LIN {X 0,Y 179.244,Z 433.398,A -85,B 0,C 180,E1 -24811.852,E2 -24811.852} C_VEL
LIN {X 0,Y 175.671,Z 428.049,A -85,B 0,C 180,E1 -24814.607,E2 -24814.607} C_VEL
LIN {X 0,Y 173.718,Z 425.111,A -85,B 0,C 180,E1 -24816.292,E2 -24816.292} C_VEL
LIN {X 0,Y 171.255,Z 421.543,A -85,B 0,C 180,E1 -24818.641,E2 -24818.641} C_VEL
LIN {X 0,Y 168.544,Z 417.832,A -85,B 0,C 180,E1 -24821.618,E2 -24821.618} C_VEL
LIN {X 0,Y 167.606,Z 416.657,A -85,B 0,C 180,E1 -24822.774,E2 -24822.774} C_VEL
LIN {X 0,Y 165.097,Z 413.195,A -85,B 0,C 180,E1 -24826.459,E2 -24826.459} C_VEL
LIN {X 0,Y 164.62,Z 412.184,A -85,B 0,C 180,E1 -24827.361,E2 -24827.361} C_VEL
LIN {X 0,Y 161.279,Z 407.116,A -85,B 0,C 180,E1 -24838.751,E2 -24838.751} C_VEL
LIN {X 0,Y 161.263,Z 406.995,A -85,B 0,C 180,E1 -24840.624,E2 -24840.624} C_VEL
LIN {X 0,Y 161.713,Z 408.835,A -85,B 0,C 180,E1 -24845.299,E2 -24845.299} C_VEL
LIN {X 0,Y 164.838,Z 412.58,A -85,B 0,C 180,E1 -24853.091,E2 -24853.091} C_VEL
LIN {X 0,Y 167.223,Z 416.316,A -85,B 0,C 180,E1 -24856.794,E2 -24856.794} C_VEL
LIN {X 0,Y 168.452,Z 417.684,A -85,B 0,C 180,E1 -24858.313,E2 -24858.313} C_VEL
LIN {X 0,Y 171.212,Z 421.521,A -85,B 0,C 180,E1 -24861.365,E2 -24861.365} C_VEL
LIN {X 0,Y 175.071,Z 427.086,A -85,B 0,C 180,E1 -24864.93,E2 -24864.93} C_VEL
LIN {X 0,Y 179.814,Z 434.296,A -85,B 0,C 180,E1 -24868.604,E2 -24868.604} C_VEL
LIN {X 0,Y 184.893,Z 442.842,A -85,B 0,C 180,E1 -24871.99,E2 -24871.99} C_VEL
LIN {X 0,Y 189.293,Z 452.81,A -85,B 0,C 180,E1 -24874.721,E2 -24874.721} C_VEL
LIN {X 0,Y 191.912,Z 459.666,A -85,B 0,C 180,E1 -24876.262,E2 -24876.262} C_VEL
LIN {X 0,Y 188.369,Z 504.662,A -85,B 0,C 180,E1 -24877.636,E2 -24877.636} C_VEL
LIN {X 0,Y 186.538,Z 518.919,A -85,B 0,C 180,E1 -24878.256,E2 -24878.256} C_VEL
LIN {X 0,Y 183.633,Z 533.235,A -85,B 0,C 180,E1 -24879.199,E2 -24879.199} C_VEL
LIN {X 0,Y 180.047,Z 546.434,A -85,B 0,C 180,E1 -24880.438,E2 -24880.438} C_VEL
LIN {X 0,Y 176.027,Z 558.458,A -85,B 0,C 180,E1 -24881.965,E2 -24881.965} C_VEL
LIN {X 0,Y 171.04,Z 570.911,A -85,B 0,C 180,E1 -24884.027,E2 -24884.027} C_VEL
LIN {X 0,Y 167.715,Z 578.171,A -85,B 0,C 180,E1 -24885.532,E2 -24885.532} C_VEL
LIN {X 0,Y 165.051,Z 582.747,A -85,B 0,C 180,E1 -24886.466,E2 -24886.466} C_VEL
LIN {X 0,Y 159.051,Z 589.893,A -85,B 0,C 180,E1 -24887.711,E2 -24887.711} C_VEL
LIN {X 0,Y 152.884,Z 596.609,A -85,B 0,C 180,E1 -24889.164,E2 -24889.164} C_VEL
LIN {X 0,Y 149.983,Z 600.384,A -85,B 0,C 180,E1 -24890.442,E2 -24890.442} C_VEL
LIN {X 0,Y 144.381,Z 608.729,A -85,B 0,C 180,E1 -24894.264,E2 -24894.264} C_VEL
LIN {X 0,Y 139.661,Z 615.209,A -85,B 0,C 180,E1 -24898.109,E2 -24898.109} C_VEL
LIN {X 0,Y 135.799,Z 620.586,A -85,B 0,C 180,E1 -24902.244,E2 -24902.244} C_VEL
LIN {X 0,Y 131.508,Z 626.247,A -85,B 0,C 180,E1 -24908.036,E2 -24908.036} C_VEL
LIN {X 0,Y 128.509,Z 630.353,A -85,B 0,C 180,E1 -24914.135,E2 -24914.135} C_VEL
LIN {X 0,Y 126.82,Z 633.026,A -85,B 0,C 180,E1 -24920.434,E2 -24920.434} C_VEL
LIN {X 0,Y 126.305,Z 634.341,A -85,B 0,C 180,E1 -24926.814,E2 -24926.814} C_VEL
LIN {X 0,Y 126.32,Z 634.5,A -85,B 0,C 180,E1 -24930.004,E2 -24930.004} C_VEL
LIN {X 0,Y 126.492,Z 633.821,A -85,B 0,C 180,E1 -24936.384,E2 -24936.384} C_VEL
LIN {X 0,Y 127.846,Z 631.805,A -85,B 0,C 180,E1 -24942.707,E2 -24942.707} C_VEL
LIN {X 0,Y 130.668,Z 628.407,A -85,B 0,C 180,E1 -24948.831,E2 -24948.831} C_VEL
LIN {X 0,Y 133.685,Z 625.344,A -85,B 0,C 180,E1 -24952.918,E2 -24952.918} C_VEL
LIN {X 0,Y 137.389,Z 628.317,A -85,B 0,C 180,E1 -24957.416,E2 -24957.416} C_VEL
LIN {X 0,Y 143.434,Z 631.102,A -85,B 0,C 180,E1 -24962.618,E2 -24962.618} C_VEL
LIN {X 0,Y 151.002,Z 632.815,A -85,B 0,C 180,E1 -24967.236,E2 -24967.236} C_VEL
LIN {X 0,Y 159.895,Z 633.459,A -85,B 0,C 180,E1 -24971.251,E2 -24971.251} C_VEL
LIN {X 0,Y 169.8,Z 633.01,A -85,B 0,C 180,E1 -24974.722,E2 -24974.722} C_VEL
LIN {X 0,Y 171.46,Z 632.84,A -85,B 0,C 180,E1 -24975.828,E2 -24975.828} C_VEL
LIN {X 0,Y 161.323,Z 633.521,A -85,B 0,C 180,E1 -24979.196,E2 -24979.196} C_VEL
LIN {X 0,Y 152.228,Z 633.038,A -85,B 0,C 180,E1 -24983.118,E2 -24983.118} C_VEL
LIN {X 0,Y 144.519,Z 631.444,A -85,B 0,C 180,E1 -24987.661,E2 -24987.661} C_VEL
LIN {X 0,Y 138.231,Z 628.727,A -85,B 0,C 180,E1 -24992.769,E2 -24992.769} C_VEL
LIN {X 0,Y 133.649,Z 624.844,A -85,B 0,C 180,E1 -24998.402,E2 -24998.402} C_VEL
LIN {X 0,Y 130.688,Z 619.649,A -85,B 0,C 180,E1 -25004.402,E2 -25004.402} C_VEL
LIN {X 0,Y 129.529,Z 613.033,A -85,B 0,C 180,E1 -25010.632,E2 -25010.632} C_VEL
LIN {X 0,Y 129.643,Z 606.868,A -85,B 0,C 180,E1 -25015.336,E2 -25015.336} C_VEL
LIN {X 0,Y 129.888,Z 600.509,A -85,B 0,C 180,E1 -25019.225,E2 -25019.225} C_VEL
LIN {X 0,Y 129.965,Z 592.706,A -85,B 0,C 180,E1 -25023.1,E2 -25023.1} C_VEL
LIN {X 0,Y 130.141,Z 583.047,A -85,B 0,C 180,E1 -25026.979,E2 -25026.979} C_VEL
LIN {X 0,Y 130.686,Z 571.183,A -85,B 0,C 180,E1 -25030.849,E2 -25030.849} C_VEL
LIN {X 0,Y 131.008,Z 565.155,A -85,B 0,C 180,E1 -25032.705,E2 -25032.705} C_VEL
LIN {X 0,Y 130.969,Z 564.229,A -85,B 0,C 180,E1 -25033.527,E2 -25033.527} C_VEL
LIN {X 0,Y 131.194,Z 564.312,A -85,B 0,C 180,E1 -25034.387,E2 -25034.387} C_VEL
LIN {X 0,Y 132.105,Z 563.892,A -85,B 0,C 180,E1 -25035.427,E2 -25035.427} C_VEL
LIN {X 0,Y 133.005,Z 563.215,A -85,B 0,C 180,E1 -25036.124,E2 -25036.124} C_VEL
LIN {X 0,Y 134.669,Z 561.654,A -85,B 0,C 180,E1 -25037.08,E2 -25037.08} C_VEL
LIN {X 0,Y 135.986,Z 560.715,A -85,B 0,C 180,E1 -25038.065,E2 -25038.065} C_VEL
LIN {X 0,Y 137.57,Z 559.906,A -85,B 0,C 180,E1 -25039.4,E2 -25039.4} C_VEL
LIN {X 0,Y 139.56,Z 558.421,A -85,B 0,C 180,E1 -25040.641,E2 -25040.641} C_VEL
LIN {X 0,Y 142.131,Z 555.895,A -85,B 0,C 180,E1 -25041.769,E2 -25041.769} C_VEL
LIN {X 0,Y 144.345,Z 554.176,A -85,B 0,C 180,E1 -25042.924,E2 -25042.924} C_VEL
LIN {X 0,Y 146.147,Z 552.999,A -85,B 0,C 180,E1 -25043.973,E2 -25043.973} C_VEL
LIN {X 0,Y 149.832,Z 549.473,A -85,B 0,C 180,E1 -25045.449,E2 -25045.449} C_VEL
LIN {X 0,Y 154.004,Z 544.288,A -85,B 0,C 180,E1 -25046.63,E2 -25046.63} C_VEL
LIN {X 0,Y 157.396,Z 541.143,A -85,B 0,C 180,E1 -25047.96,E2 -25047.96} C_VEL
LIN {X 0,Y 160.767,Z 537.171,A -85,B 0,C 180,E1 -25049.031,E2 -25049.031} C_VEL
LIN {X 0,Y 164.121,Z 532.187,A -85,B 0,C 180,E1 -25049.854,E2 -25049.854} C_VEL
LIN {X 0,Y 168.655,Z 523.446,A -85,B 0,C 180,E1 -25050.7,E2 -25050.7} C_VEL
LIN {X 0,Y 169.379,Z 522.128,A -85,B 0,C 180,E1 -25050.87,E2 -25050.87} C_VEL
LIN {X 0,Y 173.729,Z 515.688,A -85,B 0,C 180,E1 -25052.255,E2 -25052.255} C_VEL
LIN {X 0,Y 177.766,Z 507.143,A -85,B 0,C 180,E1 -25053.36,E2 -25053.36} C_VEL
LIN {X 0,Y 181.789,Z 495.234,A -85,B 0,C 180,E1 -25054.375,E2 -25054.375} C_VEL
LIN {X 0,Y 184.133,Z 487.673,A -85,B 0,C 180,E1 -25054.926,E2 -25054.926} C_VEL
LIN {X 0,Y 185.481,Z 485.476,A -85,B 0,C 180,E1 -25055.375,E2 -25055.375} C_VEL
LIN {X 0,Y 183.249,Z 510.976,A -85,B 0,C 180,E1 -25056.227,E2 -25056.227} C_VEL
LIN {X 0,Y 180.907,Z 525.142,A -85,B 0,C 180,E1 -25056.978,E2 -25056.978} C_VEL
LIN {X 0,Y 177.41,Z 539.397,A -85,B 0,C 180,E1 -25058.059,E2 -25058.059} C_VEL
LIN {X 0,Y 173.211,Z 552.958,A -85,B 0,C 180,E1 -25059.559,E2 -25059.559} C_VEL
LIN {X 0,Y 168.462,Z 565.164,A -85,B 0,C 180,E1 -25061.324,E2 -25061.324} C_VEL
LIN {X 0,Y 163.41,Z 576.407,A -85,B 0,C 180,E1 -25063.483,E2 -25063.483} C_VEL
LIN {X 0,Y 158.677,Z 585.689,A -85,B 0,C 180,E1 -25065.762,E2 -25065.762} C_VEL
LIN {X 0,Y 152.557,Z 596.127,A -85,B 0,C 180,E1 -25068.965,E2 -25068.965} C_VEL
LIN {X 0,Y 146.983,Z 604.737,A -85,B 0,C 180,E1 -25072.432,E2 -25072.432} C_VEL
LIN {X 0,Y 141.209,Z 612.989,A -85,B 0,C 180,E1 -25076.802,E2 -25076.802} C_VEL
LIN {X 0,Y 136.924,Z 618.691,A -85,B 0,C 180,E1 -25080.759,E2 -25080.759} C_VEL
LIN {X 0,Y 133.508,Z 623.478,A -85,B 0,C 180,E1 -25085.09,E2 -25085.09} C_VEL
LIN {X 0,Y 129.801,Z 628.375,A -85,B 0,C 180,E1 -25091.038,E2 -25091.038} C_VEL
LIN {X 0,Y 127.506,Z 631.784,A -85,B 0,C 180,E1 -25097.259,E2 -25097.259} C_VEL
LIN {X 0,Y 126.471,Z 633.81,A -85,B 0,C 180,E1 -25103.615,E2 -25103.615} C_VEL
LIN {X 0,Y 126.321,Z 634.499,A -85,B 0,C 180,E1 -25109.996,E2 -25109.996} C_VEL
LIN {X 0,Y 126.467,Z 633.861,A -85,B 0,C 180,E1 -25116.377,E2 -25116.377} C_VEL
LIN {X 0,Y 127.498,Z 631.882,A -85,B 0,C 180,E1 -25122.734,E2 -25122.734} C_VEL
LIN {X 0,Y 129.778,Z 628.515,A -85,B 0,C 180,E1 -25128.957,E2 -25128.957} C_VEL
LIN {X 0,Y 133.475,Z 623.659,A -85,B 0,C 180,E1 -25134.908,E2 -25134.908} C_VEL
LIN {X 0,Y 137.051,Z 618.779,A -85,B 0,C 180,E1 -25139.335,E2 -25139.335} C_VEL
LIN {X 0,Y 141.902,Z 612.177,A -85,B 0,C 180,E1 -25143.856,E2 -25143.856} C_VEL
LIN {X 0,Y 147.781,Z 603.728,A -85,B 0,C 180,E1 -25148.183,E2 -25148.183} C_VEL
LIN {X 0,Y 153.433,Z 594.914,A -85,B 0,C 180,E1 -25151.614,E2 -25151.614} C_VEL
LIN {X 0,Y 159.596,Z 584.232,A -85,B 0,C 180,E1 -25154.791,E2 -25154.791} C_VEL
LIN {X 0,Y 164.978,Z 573.429,A -85,B 0,C 180,E1 -25157.289,E2 -25157.289} C_VEL
LIN {X 0,Y 170.124,Z 561.61,A -85,B 0,C 180,E1 -25159.379,E2 -25159.379} C_VEL
LIN {X 0,Y 174.888,Z 548.55,A -85,B 0,C 180,E1 -25161.127,E2 -25161.127} C_VEL
LIN {X 0,Y 178.831,Z 534.797,A -85,B 0,C 180,E1 -25162.495,E2 -25162.495} C_VEL
LIN {X 0,Y 181.989,Z 520.199,A -85,B 0,C 180,E1 -25163.483,E2 -25163.483} C_VEL
LIN {X 0,Y 184.133,Z 505.015,A -85,B 0,C 180,E1 -25164.127,E2 -25164.127} C_VEL
LIN {X 0,Y 187.606,Z 462.246,A -85,B 0,C 180,E1 -25165.447,E2 -25165.447} C_VEL
LIN {X 0,Y 183.41,Z 451.569,A -85,B 0,C 180,E1 -25168.165,E2 -25168.165} C_VEL
LIN {X 0,Y 181.046,Z 446.597,A -85,B 0,C 180,E1 -25169.771,E2 -25169.771} C_VEL
LIN {X 0,Y 176.77,Z 439.262,A -85,B 0,C 180,E1 -25172.872,E2 -25172.872} C_VEL
LIN {X 0,Y 172.073,Z 431.836,A -85,B 0,C 180,E1 -25176.861,E2 -25176.861} C_VEL
LIN {X 0,Y 169.42,Z 427.958,A -85,B 0,C 180,E1 -25179.512,E2 -25179.512} C_VEL
LIN {X 0,Y 166.274,Z 423.469,A -85,B 0,C 180,E1 -25183.287,E2 -25183.287} C_VEL
LIN {X 0,Y 163.793,Z 419.896,A -85,B 0,C 180,E1 -25187.139,E2 -25187.139} C_VEL
LIN {X 0,Y 163.328,Z 419.049,A -85,B 0,C 180,E1 -25188.048,E2 -25188.048} C_VEL
LIN {X 0,Y 160.398,Z 414.048,A -85,B 0,C 180,E1 -25199.372,E2 -25199.372} C_VEL
LIN {X 0,Y 160.428,Z 414.414,A -85,B 0,C 180,E1 -25201.883,E2 -25201.883} C_VEL
LIN {X 0,Y 163.602,Z 419.452,A -85,B 0,C 180,E1 -25212.521,E2 -25212.521} C_VEL
LIN {X 0,Y 166.109,Z 423.331,A -85,B 0,C 180,E1 -25216.547,E2 -25216.547} C_VEL
LIN {X 0,Y 167.009,Z 424.521,A -85,B 0,C 180,E1 -25217.724,E2 -25217.724} C_VEL
LIN {X 0,Y 170.395,Z 429.368,A -85,B 0,C 180,E1 -25221.552,E2 -25221.552} C_VEL
LIN {X 0,Y 173.08,Z 433.493,A -85,B 0,C 180,E1 -25224.116,E2 -25224.116} C_VEL
LIN {X 0,Y 177.234,Z 440.033,A -85,B 0,C 180,E1 -25227.53,E2 -25227.53} C_VEL
LIN {X 0,Y 181.855,Z 448.095,A -85,B 0,C 180,E1 -25230.821,E2 -25230.821} C_VEL
LIN {X 0,Y 185.79,Z 457.378,A -85,B 0,C 180,E1 -25233.444,E2 -25233.444} C_VEL
LIN {X 0,Y 187.594,Z 462.212,A -85,B 0,C 180,E1 -25234.591,E2 -25234.591} C_VEL
LIN {X 0,Y 184.122,Z 504.68,A -85,B 0,C 180,E1 -25235.888,E2 -25235.888} C_VEL
LIN {X 0,Y 182.234,Z 518.93,A -85,B 0,C 180,E1 -25236.506,E2 -25236.506} C_VEL
LIN {X 0,Y 179.241,Z 533.243,A -85,B 0,C 180,E1 -25237.445,E2 -25237.445} C_VEL
LIN {X 0,Y 175.518,Z 546.44,A -85,B 0,C 180,E1 -25238.671,E2 -25238.671} C_VEL
LIN {X 0,Y 171.361,Z 558.463,A -85,B 0,C 180,E1 -25240.199,E2 -25240.199} C_VEL
LIN {X 0,Y 166.173,Z 570.915,A -85,B 0,C 180,E1 -25242.263,E2 -25242.263} C_VEL
LIN {X 0,Y 161.122,Z 581.495,A -85,B 0,C 180,E1 -25244.581,E2 -25244.581} C_VEL
LIN {X 0,Y 155.512,Z 591.528,A -85,B 0,C 180,E1 -25247.326,E2 -25247.326} C_VEL
LIN {X 0,Y 149.983,Z 600.384,A -85,B 0,C 180,E1 -25250.442,E2 -25250.442} C_VEL
LIN {X 0,Y 147.102,Z 604.081,A -85,B 0,C 180,E1 -25251.829,E2 -25251.829} C_VEL
LIN {X 0,Y 140.856,Z 609.711,A -85,B 0,C 180,E1 -25253.924,E2 -25253.924} C_VEL
LIN {X 0,Y 134.614,Z 614.773,A -85,B 0,C 180,E1 -25256.347,E2 -25256.347} C_VEL
LIN {X 0,Y 131.826,Z 617.572,A -85,B 0,C 180,E1 -25258.236,E2 -25258.236} C_VEL
LIN {X 0,Y 127.052,Z 623.621,A -85,B 0,C 180,E1 -25263.74,E2 -25263.74} C_VEL
LIN {X 0,Y 123.057,Z 628.487,A -85,B 0,C 180,E1 -25269.965,E2 -25269.965} C_VEL
LIN {X 0,Y 120.557,Z 631.863,A -85,B 0,C 180,E1 -25276.52,E2 -25276.52} C_VEL
LIN {X 0,Y 119.413,Z 633.851,A -85,B 0,C 180,E1 -25283.244,E2 -25283.244} C_VEL
LIN {X 0,Y 119.233,Z 634.5,A -85,B 0,C 180,E1 -25290.004,E2 -25290.004} C_VEL
LIN {X 0,Y 119.441,Z 633.821,A -85,B 0,C 180,E1 -25296.763,E2 -25296.763} C_VEL
LIN {X 0,Y 120.913,Z 631.804,A -85,B 0,C 180,E1 -25303.448,E2 -25303.448} C_VEL
LIN {X 0,Y 123.985,Z 628.404,A -85,B 0,C 180,E1 -25309.888,E2 -25309.888} C_VEL
LIN {X 0,Y 128.164,Z 624.36,A -85,B 0,C 180,E1 -25315.262,E2 -25315.262} C_VEL
LIN {X 0,Y 134.265,Z 628.587,A -85,B 0,C 180,E1 -25321.568,E2 -25321.568} C_VEL
LIN {X 0,Y 141.353,Z 631.254,A -85,B 0,C 180,E1 -25326.633,E2 -25326.633} C_VEL
LIN {X 0,Y 149.902,Z 632.893,A -85,B 0,C 180,E1 -25331.028,E2 -25331.028} C_VEL
LIN {X 0,Y 159.641,Z 633.491,A -85,B 0,C 180,E1 -25334.783,E2 -25334.783} C_VEL
LIN {X 0,Y 161.113,Z 633.483,A -85,B 0,C 180,E1 -25335.738,E2 -25335.738} C_VEL
LIN {X 0,Y 151.215,Z 633.062,A -85,B 0,C 180,E1 -25339.408,E2 -25339.408} C_VEL
LIN {X 0,Y 142.413,Z 631.536,A -85,B 0,C 180,E1 -25343.687,E2 -25343.687} C_VEL
LIN {X 0,Y 135.171,Z 628.959,A -85,B 0,C 180,E1 -25348.672,E2 -25348.672} C_VEL
LIN {X 0,Y 129.514,Z 625.273,A -85,B 0,C 180,E1 -25354.271,E2 -25354.271} C_VEL
LIN {X 0,Y 125.538,Z 620.332,A -85,B 0,C 180,E1 -25360.373,E2 -25360.373} C_VEL
LIN {X 0,Y 123.428,Z 614.039,A -85,B 0,C 180,E1 -25366.835,E2 -25366.835} C_VEL
LIN {X 0,Y 123.073,Z 607.219,A -85,B 0,C 180,E1 -25372.618,E2 -25372.618} C_VEL
LIN {X 0,Y 123.248,Z 601.253,A -85,B 0,C 180,E1 -25376.731,E2 -25376.731} C_VEL
LIN {X 0,Y 123.349,Z 595.479,A -85,B 0,C 180,E1 -25380,E2 -25380} C_VEL
LIN {X 0,Y 123.4,Z 586.697,A -85,B 0,C 180,E1 -25384.083,E2 -25384.083} C_VEL
LIN {X 0,Y 123.681,Z 574.784,A -85,B 0,C 180,E1 -25388.579,E2 -25388.579} C_VEL
LIN {X 0,Y 123.634,Z 572.839,A -85,B 0,C 180,E1 -25389.613,E2 -25389.613} C_VEL
LIN {X 0,Y 123.574,Z 572.68,A -85,B 0,C 180,E1 -25390.652,E2 -25390.652} C_VEL
LIN {X 0,Y 123.86,Z 572.688,A -85,B 0,C 180,E1 -25391.455,E2 -25391.455} C_VEL
LIN {X 0,Y 129.837,Z 569.054,A -85,B 0,C 180,E1 -25397.321,E2 -25397.321} C_VEL
LIN {X 0,Y 131.985,Z 567.401,A -85,B 0,C 180,E1 -25398.632,E2 -25398.632} C_VEL
LIN {X 0,Y 135.767,Z 565.163,A -85,B 0,C 180,E1 -25401.245,E2 -25401.245} C_VEL
LIN {X 0,Y 137.905,Z 563.714,A -85,B 0,C 180,E1 -25402.472,E2 -25402.472} C_VEL
LIN {X 0,Y 142.79,Z 559.737,A -85,B 0,C 180,E1 -25404.573,E2 -25404.573} C_VEL
LIN {X 0,Y 145.2,Z 558.222,A -85,B 0,C 180,E1 -25405.825,E2 -25405.825} C_VEL
LIN {X 0,Y 149.323,Z 554.666,A -85,B 0,C 180,E1 -25407.316,E2 -25407.316} C_VEL
LIN {X 0,Y 154.198,Z 549.261,A -85,B 0,C 180,E1 -25408.591,E2 -25408.591} C_VEL
LIN {X 0,Y 159.212,Z 544.636,A -85,B 0,C 180,E1 -25410.267,E2 -25410.267} C_VEL
LIN {X 0,Y 163.686,Z 539.253,A -85,B 0,C 180,E1 -25411.373,E2 -25411.373} C_VEL
LIN {X 0,Y 168.158,Z 532.395,A -85,B 0,C 180,E1 -25412.217,E2 -25412.217} C_VEL
LIN {X 0,Y 171.635,Z 525.96,A -85,B 0,C 180,E1 -25412.787,E2 -25412.787} C_VEL
LIN {X 0,Y 176.17,Z 519.547,A -85,B 0,C 180,E1 -25414.03,E2 -25414.03} C_VEL
LIN {X 0,Y 178.479,Z 515.409,A -85,B 0,C 180,E1 -25414.566,E2 -25414.566} C_VEL
LIN {X 0,Y 175.663,Z 529.961,A -85,B 0,C 180,E1 -25415.458,E2 -25415.458} C_VEL
LIN {X 0,Y 171.838,Z 543.659,A -85,B 0,C 180,E1 -25416.612,E2 -25416.612} C_VEL
LIN {X 0,Y 167.529,Z 556.242,A -85,B 0,C 180,E1 -25418.129,E2 -25418.129} C_VEL
LIN {X 0,Y 162.052,Z 569.104,A -85,B 0,C 180,E1 -25420.144,E2 -25420.144} C_VEL
LIN {X 0,Y 157.021,Z 579.447,A -85,B 0,C 180,E1 -25422.315,E2 -25422.315} C_VEL
LIN {X 0,Y 151.485,Z 589.388,A -85,B 0,C 180,E1 -25424.963,E2 -25424.963} C_VEL
LIN {X 0,Y 145.207,Z 599.151,A -85,B 0,C 180,E1 -25428.275,E2 -25428.275} C_VEL
LIN {X 0,Y 139.561,Z 607.25,A -85,B 0,C 180,E1 -25431.907,E2 -25431.907} C_VEL
LIN {X 0,Y 133.702,Z 615.006,A -85,B 0,C 180,E1 -25436.496,E2 -25436.496} C_VEL
LIN {X 0,Y 129.46,Z 620.426,A -85,B 0,C 180,E1 -25440.748,E2 -25440.748} C_VEL
LIN {X 0,Y 124.95,Z 626.122,A -85,B 0,C 180,E1 -25446.809,E2 -25446.809} C_VEL
LIN {X 0,Y 121.67,Z 630.258,A -85,B 0,C 180,E1 -25453.209,E2 -25453.209} C_VEL
LIN {X 0,Y 119.841,Z 632.966,A -85,B 0,C 180,E1 -25459.863,E2 -25459.863} C_VEL
LIN {X 0,Y 119.225,Z 634.321,A -85,B 0,C 180,E1 -25466.616,E2 -25466.616} C_VEL
LIN {X 0,Y 119.235,Z 634.499,A -85,B 0,C 180,E1 -25469.996,E2 -25469.996} C_VEL
LIN {X 0,Y 119.414,Z 633.86,A -85,B 0,C 180,E1 -25476.756,E2 -25476.756} C_VEL
LIN {X 0,Y 120.557,Z 631.882,A -85,B 0,C 180,E1 -25483.48,E2 -25483.48} C_VEL
LIN {X 0,Y 123.049,Z 628.514,A -85,B 0,C 180,E1 -25490.036,E2 -25490.036} C_VEL
LIN {X 0,Y 127.023,Z 623.658,A -85,B 0,C 180,E1 -25496.267,E2 -25496.267} C_VEL
LIN {X 0,Y 132.136,Z 617.168,A -85,B 0,C 180,E1 -25502.127,E2 -25502.127} C_VEL
LIN {X 0,Y 137.734,Z 609.944,A -85,B 0,C 180,E1 -25506.833,E2 -25506.833} C_VEL
LIN {X 0,Y 144.119,Z 601.005,A -85,B 0,C 180,E1 -25511.168,E2 -25511.168} C_VEL
LIN {X 0,Y 150.283,Z 591.616,A -85,B 0,C 180,E1 -25514.54,E2 -25514.54} C_VEL
LIN {X 0,Y 156.738,Z 580.323,A -85,B 0,C 180,E1 -25517.635,E2 -25517.635} C_VEL
LIN {X 0,Y 162.586,Z 568.458,A -85,B 0,C 180,E1 -25520.104,E2 -25520.104} C_VEL
LIN {X 0,Y 167.422,Z 557.033,A -85,B 0,C 180,E1 -25521.908,E2 -25521.908} C_VEL
LIN {X 0,Y 171.752,Z 544.64,A -85,B 0,C 180,E1 -25523.416,E2 -25523.416} C_VEL
LIN {X 0,Y 175.576,Z 530.887,A -85,B 0,C 180,E1 -25524.639,E2 -25524.639} C_VEL
LIN {X 0,Y 178.539,Z 516.529,A -85,B 0,C 180,E1 -25525.5,E2 -25525.5} C_VEL
LIN {X 0,Y 180.311,Z 502.555,A -85,B 0,C 180,E1 -25526.043,E2 -25526.043} C_VEL
LIN {X 0,Y 183.397,Z 465.809,A -85,B 0,C 180,E1 -25527.151,E2 -25527.151} C_VEL
LIN {X 0,Y 183.298,Z 464.508,A -85,B 0,C 180,E1 -25527.291,E2 -25527.291} C_VEL
LIN {X 0,Y 179.876,Z 455.579,A -85,B 0,C 180,E1 -25529.713,E2 -25529.713} C_VEL
LIN {X 0,Y 177.842,Z 451.275,A -85,B 0,C 180,E1 -25531.204,E2 -25531.204} C_VEL
LIN {X 0,Y 173.619,Z 443.994,A -85,B 0,C 180,E1 -25534.526,E2 -25534.526} C_VEL
LIN {X 0,Y 170.002,Z 437.971,A -85,B 0,C 180,E1 -25537.868,E2 -25537.868} C_VEL
LIN {X 0,Y 167.626,Z 434.367,A -85,B 0,C 180,E1 -25540.402,E2 -25540.402} C_VEL
LIN {X 0,Y 164.838,Z 430.147,A -85,B 0,C 180,E1 -25543.971,E2 -25543.971} C_VEL
LIN {X 0,Y 162.44,Z 426.442,A -85,B 0,C 180,E1 -25547.982,E2 -25547.982} C_VEL
LIN {X 0,Y 161.615,Z 425.498,A -85,B 0,C 180,E1 -25549.666,E2 -25549.666} C_VEL
LIN {X 0,Y 159.53,Z 421.118,A -85,B 0,C 180,E1 -25559.369,E2 -25559.369} C_VEL
LIN {X 0,Y 159.543,Z 421.41,A -85,B 0,C 180,E1 -25561.577,E2 -25561.577} C_VEL
LIN {X 0,Y 162.35,Z 426.213,A -85,B 0,C 180,E1 -25571.866,E2 -25571.866} C_VEL
LIN {X 0,Y 164.77,Z 430.115,A -85,B 0,C 180,E1 -25575.987,E2 -25575.987} C_VEL
LIN {X 0,Y 165.942,Z 431.936,A -85,B 0,C 180,E1 -25577.603,E2 -25577.603} C_VEL
LIN {X 0,Y 168.626,Z 435.83,A -85,B 0,C 180,E1 -25580.748,E2 -25580.748} C_VEL
LIN {X 0,Y 171.216,Z 440.009,A -85,B 0,C 180,E1 -25583.366,E2 -25583.366} C_VEL
LIN {X 0,Y 175.168,Z 446.566,A -85,B 0,C 180,E1 -25586.791,E2 -25586.791} C_VEL
LIN {X 0,Y 179.146,Z 453.795,A -85,B 0,C 180,E1 -25589.789,E2 -25589.789} C_VEL
LIN {X 0,Y 182.975,Z 463.573,A -85,B 0,C 180,E1 -25592.529,E2 -25592.529} C_VEL
LIN {X 0,Y 183.423,Z 464.819,A -85,B 0,C 180,E1 -25592.837,E2 -25592.837} C_VEL
LIN {X 0,Y 180.512,Z 499.873,A -85,B 0,C 180,E1 -25593.909,E2 -25593.909} C_VEL
LIN {X 0,Y 178.944,Z 514.023,A -85,B 0,C 180,E1 -25594.44,E2 -25594.44} C_VEL
LIN {X 0,Y 176.346,Z 527.897,A -85,B 0,C 180,E1 -25595.221,E2 -25595.221} C_VEL
LIN {X 0,Y 172.786,Z 541.436,A -85,B 0,C 180,E1 -25596.312,E2 -25596.312} C_VEL
LIN {X 0,Y 168.684,Z 553.682,A -85,B 0,C 180,E1 -25597.669,E2 -25597.669} C_VEL
LIN {X 0,Y 163.837,Z 565.741,A -85,B 0,C 180,E1 -25599.46,E2 -25599.46} C_VEL
LIN {X 0,Y 157.846,Z 578.188,A -85,B 0,C 180,E1 -25601.903,E2 -25601.903} C_VEL
LIN {X 0,Y 152.524,Z 587.969,A -85,B 0,C 180,E1 -25604.427,E2 -25604.427} C_VEL
LIN {X 0,Y 146.171,Z 597.967,A -85,B 0,C 180,E1 -25607.696,E2 -25607.696} C_VEL
LIN {X 0,Y 140.434,Z 606.268,A -85,B 0,C 180,E1 -25611.282,E2 -25611.282} C_VEL
LIN {X 0,Y 134.435,Z 614.204,A -85,B 0,C 180,E1 -25615.812,E2 -25615.812} C_VEL
LIN {X 0,Y 131.826,Z 617.572,A -85,B 0,C 180,E1 -25618.236,E2 -25618.236} C_VEL
LIN {X 0,Y 129.149,Z 620.212,A -85,B 0,C 180,E1 -25620.25,E2 -25620.25} C_VEL
LIN {X 0,Y 121.061,Z 625.462,A -85,B 0,C 180,E1 -25624.844,E2 -25624.844} C_VEL
LIN {X 0,Y 117.141,Z 627.938,A -85,B 0,C 180,E1 -25627.939,E2 -25627.939} C_VEL
LIN {X 0,Y 115.916,Z 629.007,A -85,B 0,C 180,E1 -25629.707,E2 -25629.707} C_VEL
LIN {X 0,Y 113.647,Z 631.863,A -85,B 0,C 180,E1 -25635.683,E2 -25635.683} C_VEL
LIN {X 0,Y 112.337,Z 633.851,A -85,B 0,C 180,E1 -25642.817,E2 -25642.817} C_VEL
LIN {X 0,Y 112.133,Z 634.341,A -85,B 0,C 180,E1 -25646.411,E2 -25646.411} C_VEL
LIN {X 0,Y 112.139,Z 634.5,A -85,B 0,C 180,E1 -25650.005,E2 -25650.005} C_VEL
LIN {X 0,Y 112.378,Z 633.82,A -85,B 0,C 180,E1 -25657.19,E2 -25657.19} C_VEL
LIN {X 0,Y 114.013,Z 631.804,A -85,B 0,C 180,E1 -25664.279,E2 -25664.279} C_VEL
LIN {X 0,Y 117.334,Z 628.402,A -85,B 0,C 180,E1 -25671.067,E2 -25671.067} C_VEL
LIN {X 0,Y 122.927,Z 623.35,A -85,B 0,C 180,E1 -25677.8,E2 -25677.8} C_VEL
LIN {X 0,Y 128.411,Z 627.087,A -85,B 0,C 180,E1 -25683.187,E2 -25683.187} C_VEL
LIN {X 0,Y 135.788,Z 630.172,A -85,B 0,C 180,E1 -25688.4,E2 -25688.4} C_VEL
LIN {X 0,Y 144.655,Z 632.266,A -85,B 0,C 180,E1 -25692.862,E2 -25692.862} C_VEL
LIN {X 0,Y 149.529,Z 632.937,A -85,B 0,C 180,E1 -25694.835,E2 -25694.835} C_VEL
LIN {X 0,Y 150.87,Z 633.06,A -85,B 0,C 180,E1 -25695.674,E2 -25695.674} C_VEL
LIN {X 0,Y 141.194,Z 631.592,A -85,B 0,C 180,E1 -25699.678,E2 -25699.678} C_VEL
LIN {X 0,Y 132.9,Z 629.096,A -85,B 0,C 180,E1 -25704.43,E2 -25704.43} C_VEL
LIN {X 0,Y 126.114,Z 625.543,A -85,B 0,C 180,E1 -25709.898,E2 -25709.898} C_VEL
LIN {X 0,Y 121.109,Z 620.87,A -85,B 0,C 180,E1 -25716.033,E2 -25716.033} C_VEL
LIN {X 0,Y 117.55,Z 613.744,A -85,B 0,C 180,E1 -25723.78,E2 -25723.78} C_VEL
LIN {X 0,Y 116.657,Z 606.344,A -85,B 0,C 180,E1 -25730.464,E2 -25730.464} C_VEL
LIN {X 0,Y 116.799,Z 600.442,A -85,B 0,C 180,E1 -25734.822,E2 -25734.822} C_VEL
LIN {X 0,Y 116.878,Z 593.19,A -85,B 0,C 180,E1 -25739.139,E2 -25739.139} C_VEL
LIN {X 0,Y 116.843,Z 585.122,A -85,B 0,C 180,E1 -25743.017,E2 -25743.017} C_VEL
LIN {X 0,Y 116.745,Z 580.735,A -85,B 0,C 180,E1 -25745.073,E2 -25745.073} C_VEL
LIN {X 0,Y 116.491,Z 580.022,A -85,B 0,C 180,E1 -25746.061,E2 -25746.061} C_VEL
LIN {X 0,Y 116.434,Z 580.169,A -85,B 0,C 180,E1 -25746.934,E2 -25746.934} C_VEL
LIN {X 0,Y 118.707,Z 578.589,A -85,B 0,C 180,E1 -25750.231,E2 -25750.231} C_VEL
LIN {X 0,Y 120.82,Z 577.705,A -85,B 0,C 180,E1 -25753.455,E2 -25753.455} C_VEL
LIN {X 0,Y 127.517,Z 574.056,A -85,B 0,C 180,E1 -25759.311,E2 -25759.311} C_VEL
LIN {X 0,Y 129.817,Z 572.488,A -85,B 0,C 180,E1 -25760.604,E2 -25760.604} C_VEL
LIN {X 0,Y 132.976,Z 570.825,A -85,B 0,C 180,E1 -25762.637,E2 -25762.637} C_VEL
LIN {X 0,Y 136.203,Z 568.867,A -85,B 0,C 180,E1 -25764.381,E2 -25764.381} C_VEL
LIN {X 0,Y 141.611,Z 564.89,A -85,B 0,C 180,E1 -25766.53,E2 -25766.53} C_VEL
LIN {X 0,Y 143.96,Z 563.522,A -85,B 0,C 180,E1 -25767.632,E2 -25767.632} C_VEL
LIN {X 0,Y 148.791,Z 559.745,A -85,B 0,C 180,E1 -25769.228,E2 -25769.228} C_VEL
LIN {X 0,Y 154.907,Z 553.647,A -85,B 0,C 180,E1 -25770.691,E2 -25770.691} C_VEL
LIN {X 0,Y 160.305,Z 548.921,A -85,B 0,C 180,E1 -25772.26,E2 -25772.26} C_VEL
LIN {X 0,Y 165.839,Z 542.606,A -85,B 0,C 180,E1 -25773.43,E2 -25773.43} C_VEL
LIN {X 0,Y 169.708,Z 537.153,A -85,B 0,C 180,E1 -25774.076,E2 -25774.076} C_VEL
LIN {X 0,Y 165.817,Z 549.44,A -85,B 0,C 180,E1 -25775.32,E2 -25775.32} C_VEL
LIN {X 0,Y 160.697,Z 562.322,A -85,B 0,C 180,E1 -25777.041,E2 -25777.041} C_VEL
LIN {X 0,Y 155.154,Z 574.017,A -85,B 0,C 180,E1 -25779.126,E2 -25779.126} C_VEL
LIN {X 0,Y 149.974,Z 583.745,A -85,B 0,C 180,E1 -25781.424,E2 -25781.424} C_VEL
LIN {X 0,Y 143.212,Z 594.505,A -85,B 0,C 180,E1 -25784.632,E2 -25784.632} C_VEL
LIN {X 0,Y 136.957,Z 603.388,A -85,B 0,C 180,E1 -25788.152,E2 -25788.152} C_VEL
LIN {X 0,Y 130.381,Z 611.895,A -85,B 0,C 180,E1 -25792.665,E2 -25792.665} C_VEL
LIN {X 0,Y 123.987,Z 619.507,A -85,B 0,C 180,E1 -25798.239,E2 -25798.239} C_VEL
LIN {X 0,Y 119.544,Z 624.882,A -85,B 0,C 180,E1 -25803.833,E2 -25803.833} C_VEL
LIN {X 0,Y 116.401,Z 628.376,A -85,B 0,C 180,E1 -25808.756,E2 -25808.756} C_VEL
LIN {X 0,Y 113.654,Z 631.786,A -85,B 0,C 180,E1 -25815.675,E2 -25815.675} C_VEL
LIN {X 0,Y 112.346,Z 633.81,A -85,B 0,C 180,E1 -25822.808,E2 -25822.808} C_VEL
LIN {X 0,Y 112.135,Z 634.321,A -85,B 0,C 180,E1 -25826.402,E2 -25826.402} C_VEL
LIN {X 0,Y 112.14,Z 634.499,A -85,B 0,C 180,E1 -25829.995,E2 -25829.995} C_VEL
LIN {X 0,Y 112.134,Z 634.345,A -85,B 0,C 180,E1 -25833.589,E2 -25833.589} C_VEL
LIN {X 0,Y 112.798,Z 633.041,A -85,B 0,C 180,E1 -25840.768,E2 -25840.768} C_VEL
LIN {X 0,Y 114.848,Z 630.376,A -85,B 0,C 180,E1 -25847.812,E2 -25847.812} C_VEL
LIN {X 0,Y 118.391,Z 626.279,A -85,B 0,C 180,E1 -25854.548,E2 -25854.548} C_VEL
LIN {X 0,Y 123.253,Z 620.627,A -85,B 0,C 180,E1 -25860.871,E2 -25860.871} C_VEL
LIN {X 0,Y 128.576,Z 614.252,A -85,B 0,C 180,E1 -25865.981,E2 -25865.981} C_VEL
LIN {X 0,Y 134.883,Z 606.327,A -85,B 0,C 180,E1 -25870.635,E2 -25870.635} C_VEL
LIN {X 0,Y 140.93,Z 598.036,A -85,B 0,C 180,E1 -25874.274,E2 -25874.274} C_VEL
LIN {X 0,Y 147.554,Z 588.051,A -85,B 0,C 180,E1 -25877.578,E2 -25877.578} C_VEL
LIN {X 0,Y 153.5,Z 577.652,A -85,B 0,C 180,E1 -25880.241,E2 -25880.241} C_VEL
LIN {X 0,Y 159.363,Z 565.863,A -85,B 0,C 180,E1 -25882.537,E2 -25882.537} C_VEL
LIN {X 0,Y 164.423,Z 553.835,A -85,B 0,C 180,E1 -25884.298,E2 -25884.298} C_VEL
LIN {X 0,Y 168.943,Z 540.509,A -85,B 0,C 180,E1 -25885.765,E2 -25885.765} C_VEL
LIN {X 0,Y 172.407,Z 527.403,A -85,B 0,C 180,E1 -25886.812,E2 -25886.812} C_VEL
LIN {X 0,Y 175.068,Z 513.664,A -85,B 0,C 180,E1 -25887.544,E2 -25887.544} C_VEL
LIN {X 0,Y 177.056,Z 495.375,A -85,B 0,C 180,E1 -25888.176,E2 -25888.176} C_VEL
LIN {X 0,Y 179.477,Z 467.654,A -85,B 0,C 180,E1 -25889.001,E2 -25889.001} C_VEL
LIN {X 0,Y 176.177,Z 458.866,A -85,B 0,C 180,E1 -25891.562,E2 -25891.562} C_VEL
LIN {X 0,Y 172.155,Z 451.258,A -85,B 0,C 180,E1 -25894.86,E2 -25894.86} C_VEL
LIN {X 0,Y 168.032,Z 444.135,A -85,B 0,C 180,E1 -25898.854,E2 -25898.854} C_VEL
LIN {X 0,Y 165.875,Z 440.755,A -85,B 0,C 180,E1 -25901.312,E2 -25901.312} C_VEL
LIN {X 0,Y 163.439,Z 436.867,A -85,B 0,C 180,E1 -25904.643,E2 -25904.643} C_VEL
LIN {X 0,Y 160.904,Z 432.72,A -85,B 0,C 180,E1 -25909.302,E2 -25909.302} C_VEL
LIN {X 0,Y 158.662,Z 428.191,A -85,B 0,C 180,E1 -25919.365,E2 -25919.365} C_VEL
LIN {X 0,Y 158.662,Z 428.409,A -85,B 0,C 180,E1 -25921.269,E2 -25921.269} C_VEL
LIN {X 0,Y 161.237,Z 433.261,A -85,B 0,C 180,E1 -25931.471,E2 -25931.471} C_VEL
LIN {X 0,Y 164.113,Z 437.963,A -85,B 0,C 180,E1 -25936.403,E2 -25936.403} C_VEL
LIN {X 0,Y 167.011,Z 442.547,A -85,B 0,C 180,E1 -25940.073,E2 -25940.073} C_VEL
LIN {X 0,Y 169.352,Z 446.473,A -85,B 0,C 180,E1 -25942.57,E2 -25942.57} C_VEL
LIN {X 0,Y 172.923,Z 452.666,A -85,B 0,C 180,E1 -25945.852,E2 -25945.852} C_VEL
LIN {X 0,Y 176.385,Z 459.321,A -85,B 0,C 180,E1 -25948.645,E2 -25948.645} C_VEL
LIN {X 0,Y 179.441,Z 467.549,A -85,B 0,C 180,E1 -25951.018,E2 -25951.018} C_VEL
LIN {X 0,Y 176.549,Z 501.115,A -85,B 0,C 180,E1 -25952.037,E2 -25952.037} C_VEL
LIN {X 0,Y 174.698,Z 516.208,A -85,B 0,C 180,E1 -25952.622,E2 -25952.622} C_VEL
LIN {X 0,Y 171.686,Z 530.659,A -85,B 0,C 180,E1 -25953.488,E2 -25953.488} C_VEL
LIN {X 0,Y 168.359,Z 542.475,A -85,B 0,C 180,E1 -25954.474,E2 -25954.474} C_VEL
LIN {X 0,Y 163.804,Z 555.31,A -85,B 0,C 180,E1 -25955.927,E2 -25955.927} C_VEL
LIN {X 0,Y 158.793,Z 567.051,A -85,B 0,C 180,E1 -25957.715,E2 -25957.715} C_VEL
LIN {X 0,Y 152.744,Z 578.981,A -85,B 0,C 180,E1 -25960.103,E2 -25960.103} C_VEL
LIN {X 0,Y 147.635,Z 587.972,A -85,B 0,C 180,E1 -25962.456,E2 -25962.456} C_VEL
LIN {X 0,Y 140.99,Z 597.969,A -85,B 0,C 180,E1 -25965.75,E2 -25965.75} C_VEL
LIN {X 0,Y 134.95,Z 606.27,A -85,B 0,C 180,E1 -25969.39,E2 -25969.39} C_VEL
LIN {X 0,Y 128.59,Z 614.206,A -85,B 0,C 180,E1 -25974.023,E2 -25974.023} C_VEL
LIN {X 0,Y 123.299,Z 620.589,A -85,B 0,C 180,E1 -25979.141,E2 -25979.141} C_VEL
LIN {X 0,Y 118.408,Z 626.249,A -85,B 0,C 180,E1 -25985.455,E2 -25985.455} C_VEL
LIN {X 0,Y 115.916,Z 629.007,A -85,B 0,C 180,E1 -25989.707,E2 -25989.707} C_VEL
LIN {X 0,Y 114.072,Z 630.522,A -85,B 0,C 180,E1 -25992.412,E2 -25992.412} C_VEL
LIN {X 0,Y 109.757,Z 632.413,A -85,B 0,C 180,E1 -25996.878,E2 -25996.878} C_VEL
LIN {X 0,Y 106.574,Z 633.493,A -85,B 0,C 180,E1 -26000.709,E2 -26000.709} C_VEL
LIN {X 0,Y 105.209,Z 634.056,A -85,B 0,C 180,E1 -26003.821,E2 -26003.821} C_VEL
LIN {X 0,Y 105.069,Z 634.179,A -85,B 0,C 180,E1 -26004.894,E2 -26004.894} C_VEL
LIN {X 0,Y 105.038,Z 634.5,A -85,B 0,C 180,E1 -26010.005,E2 -26010.005} C_VEL
LIN {X 0,Y 105.324,Z 633.82,A -85,B 0,C 180,E1 -26017.674,E2 -26017.674} C_VEL
LIN {X 0,Y 107.148,Z 631.803,A -85,B 0,C 180,E1 -26025.215,E2 -26025.215} C_VEL
LIN {X 0,Y 110.743,Z 628.402,A -85,B 0,C 180,E1 -26032.386,E2 -26032.386} C_VEL
LIN {X 0,Y 114.625,Z 624.912,A -85,B 0,C 180,E1 -26037.382,E2 -26037.382} C_VEL
LIN {X 0,Y 118.146,Z 622.158,A -85,B 0,C 180,E1 -26040.625,E2 -26040.625} C_VEL
LIN {X 0,Y 126.339,Z 627.203,A -85,B 0,C 180,E1 -26047.732,E2 -26047.732} C_VEL
LIN {X 0,Y 134.81,Z 630.228,A -85,B 0,C 180,E1 -26052.671,E2 -26052.671} C_VEL
LIN {X 0,Y 139.574,Z 631.386,A -85,B 0,C 180,E1 -26054.83,E2 -26054.83} C_VEL
LIN {X 0,Y 140.81,Z 631.616,A -85,B 0,C 180,E1 -26055.673,E2 -26055.673} C_VEL
LIN {X 0,Y 131.419,Z 629.155,A -85,B 0,C 180,E1 -26060.079,E2 -26060.079} C_VEL
LIN {X 0,Y 123.594,Z 625.714,A -85,B 0,C 180,E1 -26065.345,E2 -26065.345} C_VEL
LIN {X 0,Y 117.42,Z 621.204,A -85,B 0,C 180,E1 -26071.391,E2 -26071.391} C_VEL
LIN {X 0,Y 113.081,Z 615.497,A -85,B 0,C 180,E1 -26078.106,E2 -26078.106} C_VEL
LIN {X 0,Y 110.612,Z 607.361,A -85,B 0,C 180,E1 -26086.216,E2 -26086.216} C_VEL
LIN {X 0,Y 110.445,Z 599.498,A -85,B 0,C 180,E1 -26092.689,E2 -26092.689} C_VEL
LIN {X 0,Y 110.537,Z 592.404,A -85,B 0,C 180,E1 -26097.267,E2 -26097.267} C_VEL
LIN {X 0,Y 110.284,Z 587.275,A -85,B 0,C 180,E1 -26100.229,E2 -26100.229} C_VEL
LIN {X 0,Y 109.898,Z 586.748,A -85,B 0,C 180,E1 -26101.374,E2 -26101.374} C_VEL
LIN {X 0,Y 110.041,Z 586.727,A -85,B 0,C 180,E1 -26103.662,E2 -26103.662} C_VEL
LIN {X 0,Y 114.948,Z 583.741,A -85,B 0,C 180,E1 -26111.953,E2 -26111.953} C_VEL
LIN {X 0,Y 116.365,Z 583.216,A -85,B 0,C 180,E1 -26113.98,E2 -26113.98} C_VEL
LIN {X 0,Y 123.152,Z 579.936,A -85,B 0,C 180,E1 -26120.024,E2 -26120.024} C_VEL
LIN {X 0,Y 125.171,Z 578.903,A -85,B 0,C 180,E1 -26121.405,E2 -26121.405} C_VEL
LIN {X 0,Y 127.615,Z 577.443,A -85,B 0,C 180,E1 -26122.675,E2 -26122.675} C_VEL
LIN {X 0,Y 134.479,Z 573.878,A -85,B 0,C 180,E1 -26126.374,E2 -26126.374} C_VEL
LIN {X 0,Y 140.179,Z 570.037,A -85,B 0,C 180,E1 -26128.444,E2 -26128.444} C_VEL
LIN {X 0,Y 144.13,Z 567.714,A -85,B 0,C 180,E1 -26129.988,E2 -26129.988} C_VEL
LIN {X 0,Y 150.043,Z 563.174,A -85,B 0,C 180,E1 -26131.633,E2 -26131.633} C_VEL
LIN {X 0,Y 155.656,Z 557.974,A -85,B 0,C 180,E1 -26132.807,E2 -26132.807} C_VEL
LIN {X 0,Y 159.134,Z 555.204,A -85,B 0,C 180,E1 -26133.717,E2 -26133.717} C_VEL
LIN {X 0,Y 159.005,Z 556.63,A -85,B 0,C 180,E1 -26134.16,E2 -26134.16} C_VEL
LIN {X 0,Y 153.281,Z 569.113,A -85,B 0,C 180,E1 -26136.083,E2 -26136.083} C_VEL
LIN {X 0,Y 146.973,Z 580.929,A -85,B 0,C 180,E1 -26138.578,E2 -26138.578} C_VEL
LIN {X 0,Y 140.622,Z 591.175,A -85,B 0,C 180,E1 -26141.434,E2 -26141.434} C_VEL
LIN {X 0,Y 133.827,Z 600.641,A -85,B 0,C 180,E1 -26144.845,E2 -26144.845} C_VEL
LIN {X 0,Y 126.692,Z 609.665,A -85,B 0,C 180,E1 -26149.317,E2 -26149.317} C_VEL
LIN {X 0,Y 120.315,Z 616.943,A -85,B 0,C 180,E1 -26154.253,E2 -26154.253} C_VEL
LIN {X 0,Y 115.777,Z 622.04,A -85,B 0,C 180,E1 -26158.933,E2 -26158.933} C_VEL
LIN {X 0,Y 111.985,Z 626.124,A -85,B 0,C 180,E1 -26163.935,E2 -26163.935} C_VEL
LIN {X 0,Y 108.079,Z 630.26,A -85,B 0,C 180,E1 -26171.022,E2 -26171.022} C_VEL
LIN {X 0,Y 105.839,Z 632.967,A -85,B 0,C 180,E1 -26178.504,E2 -26178.504} C_VEL
LIN {X 0,Y 105.045,Z 634.321,A -85,B 0,C 180,E1 -26186.159,E2 -26186.159} C_VEL
LIN {X 0,Y 105.039,Z 634.499,A -85,B 0,C 180,E1 -26189.995,E2 -26189.995} C_VEL
LIN {X 0,Y 105.044,Z 634.345,A -85,B 0,C 180,E1 -26193.831,E2 -26193.831} C_VEL
LIN {X 0,Y 105.817,Z 633.04,A -85,B 0,C 180,E1 -26201.488,E2 -26201.488} C_VEL
LIN {X 0,Y 108.063,Z 630.375,A -85,B 0,C 180,E1 -26208.971,E2 -26208.971} C_VEL
LIN {X 0,Y 111.951,Z 626.278,A -85,B 0,C 180,E1 -26216.063,E2 -26216.063} C_VEL
LIN {X 0,Y 117.181,Z 620.626,A -85,B 0,C 180,E1 -26222.663,E2 -26222.663} C_VEL
LIN {X 0,Y 122.882,Z 614.251,A -85,B 0,C 180,E1 -26227.934,E2 -26227.934} C_VEL
LIN {X 0,Y 129.563,Z 606.325,A -85,B 0,C 180,E1 -26232.685,E2 -26232.685} C_VEL
LIN {X 0,Y 135.937,Z 598.034,A -85,B 0,C 180,E1 -26236.364,E2 -26236.364} C_VEL
LIN {X 0,Y 142.846,Z 588.048,A -85,B 0,C 180,E1 -26239.688,E2 -26239.688} C_VEL
LIN {X 0,Y 149.465,Z 576.926,A -85,B 0,C 180,E1 -26242.506,E2 -26242.506} C_VEL
LIN {X 0,Y 155.145,Z 565.858,A -85,B 0,C 180,E1 -26244.619,E2 -26244.619} C_VEL
LIN {X 0,Y 160.393,Z 553.83,A -85,B 0,C 180,E1 -26246.353,E2 -26246.353} C_VEL
LIN {X 0,Y 165.056,Z 540.501,A -85,B 0,C 180,E1 -26247.801,E2 -26247.801} C_VEL
LIN {X 0,Y 168.637,Z 527.393,A -85,B 0,C 180,E1 -26248.825,E2 -26248.825} C_VEL
LIN {X 0,Y 171.445,Z 513.065,A -85,B 0,C 180,E1 -26249.575,E2 -26249.575} C_VEL
LIN {X 0,Y 173.388,Z 495.753,A -85,B 0,C 180,E1 -26250.154,E2 -26250.154} C_VEL
LIN {X 0,Y 175.663,Z 470.361,A -85,B 0,C 180,E1 -26250.912,E2 -26250.912} C_VEL
LIN {X 0,Y 173.115,Z 463.546,A -85,B 0,C 180,E1 -26253.069,E2 -26253.069} C_VEL
LIN {X 0,Y 169.638,Z 456.772,A -85,B 0,C 180,E1 -26256.165,E2 -26256.165} C_VEL
LIN {X 0,Y 166.252,Z 450.557,A -85,B 0,C 180,E1 -26259.702,E2 -26259.702} C_VEL
LIN {X 0,Y 164.052,Z 446.99,A -85,B 0,C 180,E1 -26262.388,E2 -26262.388} C_VEL
LIN {X 0,Y 162.019,Z 443.524,A -85,B 0,C 180,E1 -26265.396,E2 -26265.396} C_VEL
LIN {X 0,Y 159.753,Z 439.615,A -85,B 0,C 180,E1 -26269.865,E2 -26269.865} C_VEL
LIN {X 0,Y 157.799,Z 435.133,A -85,B 0,C 180,E1 -26280,E2 -26280} C_VEL
LIN {X 0,Y 160.038,Z 440.047,A -85,B 0,C 180,E1 -26290.836,E2 -26290.836} C_VEL
LIN {X 0,Y 162.726,Z 444.73,A -85,B 0,C 180,E1 -26295.767,E2 -26295.767} C_VEL
LIN {X 0,Y 165.306,Z 449,A -85,B 0,C 180,E1 -26299.238,E2 -26299.238} C_VEL
LIN {X 0,Y 168.445,Z 454.479,A -85,B 0,C 180,E1 -26302.698,E2 -26302.698} C_VEL
LIN {X 0,Y 172.59,Z 462.428,A -85,B 0,C 180,E1 -26306.529,E2 -26306.529} C_VEL
LIN {X 0,Y 174.506,Z 467.05,A -85,B 0,C 180,E1 -26308.161,E2 -26308.161} C_VEL
LIN {X 0,Y 175.643,Z 470.311,A -85,B 0,C 180,E1 -26309.117,E2 -26309.117} C_VEL
LIN {X 0,Y 172.946,Z 500.508,A -85,B 0,C 180,E1 -26310.025,E2 -26310.025} C_VEL
LIN {X 0,Y 171.108,Z 515.536,A -85,B 0,C 180,E1 -26310.594,E2 -26310.594} C_VEL
LIN {X 0,Y 168.226,Z 529.366,A -85,B 0,C 180,E1 -26311.377,E2 -26311.377} C_VEL
LIN {X 0,Y 164.449,Z 542.482,A -85,B 0,C 180,E1 -26312.437,E2 -26312.437} C_VEL
LIN {X 0,Y 159.737,Z 555.315,A -85,B 0,C 180,E1 -26313.862,E2 -26313.862} C_VEL
LIN {X 0,Y 154.546,Z 567.055,A -85,B 0,C 180,E1 -26315.629,E2 -26315.629} C_VEL
LIN {X 0,Y 148.423,Z 578.725,A -85,B 0,C 180,E1 -26317.946,E2 -26317.946} C_VEL
LIN {X 0,Y 141.752,Z 589.755,A -85,B 0,C 180,E1 -26320.885,E2 -26320.885} C_VEL
LIN {X 0,Y 134.89,Z 599.456,A -85,B 0,C 180,E1 -26324.248,E2 -26324.248} C_VEL
LIN {X 0,Y 128.609,Z 607.503,A -85,B 0,C 180,E1 -26327.984,E2 -26327.984} C_VEL
LIN {X 0,Y 122.008,Z 615.214,A -85,B 0,C 180,E1 -26332.789,E2 -26332.789} C_VEL
LIN {X 0,Y 117.215,Z 620.59,A -85,B 0,C 180,E1 -26337.348,E2 -26337.348} C_VEL
LIN {X 0,Y 111.968,Z 626.25,A -85,B 0,C 180,E1 -26343.941,E2 -26343.941} C_VEL
LIN {X 0,Y 108.067,Z 630.355,A -85,B 0,C 180,E1 -26351.029,E2 -26351.029} C_VEL
LIN {X 0,Y 105.816,Z 633.027,A -85,B 0,C 180,E1 -26358.512,E2 -26358.512} C_VEL
LIN {X 0,Y 105.069,Z 634.179,A -85,B 0,C 180,E1 -26364.894,E2 -26364.894} C_VEL
LIN {X 0,Y 104.287,Z 634.484,A -85,B 0,C 180,E1 -26368.089,E2 -26368.089} C_VEL
LIN {X 0,Y 102.67,Z 634.568,A -85,B 0,C 180,E1 -26371.26,E2 -26371.26} C_VEL
LIN {X 0,Y 99.361,Z 633.986,A -85,B 0,C 180,E1 -26377.818,E2 -26377.818} C_VEL
LIN {X 0,Y 98.898,Z 633.265,A -85,B 0,C 180,E1 -26381.245,E2 -26381.245} C_VEL
LIN {X 0,Y 99.079,Z 632.954,A -85,B 0,C 180,E1 -26382.382,E2 -26382.382} C_VEL
LIN {X 0,Y 101.977,Z 630.28,A -85,B 0,C 180,E1 -26390.162,E2 -26390.162} C_VEL
LIN {X 0,Y 106.826,Z 626.151,A -85,B 0,C 180,E1 -26397.426,E2 -26397.426} C_VEL
LIN {X 0,Y 113.546,Z 620.953,A -85,B 0,C 180,E1 -26403.591,E2 -26403.591} C_VEL
LIN {X 0,Y 120.981,Z 625.402,A -85,B 0,C 180,E1 -26409.723,E2 -26409.723} C_VEL
LIN {X 0,Y 129.78,Z 628.863,A -85,B 0,C 180,E1 -26414.753,E2 -26414.753} C_VEL
LIN {X 0,Y 130.849,Z 629.167,A -85,B 0,C 180,E1 -26415.714,E2 -26415.714} C_VEL
LIN {X 0,Y 121.953,Z 625.793,A -85,B 0,C 180,E1 -26420.66,E2 -26420.66} C_VEL
LIN {X 0,Y 114.601,Z 621.402,A -85,B 0,C 180,E1 -26426.501,E2 -26426.501} C_VEL
LIN {X 0,Y 109.097,Z 615.923,A -85,B 0,C 180,E1 -26433.196,E2 -26433.196} C_VEL
LIN {X 0,Y 105.557,Z 609.133,A -85,B 0,C 180,E1 -26440.555,E2 -26440.555} C_VEL
LIN {X 0,Y 104.267,Z 600.771,A -85,B 0,C 180,E1 -26448.334,E2 -26448.334} C_VEL
LIN {X 0,Y 104.141,Z 594.039,A -85,B 0,C 180,E1 -26453.704,E2 -26453.704} C_VEL
LIN {X 0,Y 103.693,Z 593.334,A -85,B 0,C 180,E1 -26455.14,E2 -26455.14} C_VEL
LIN {X 0,Y 103.455,Z 593.349,A -85,B 0,C 180,E1 -26456.105,E2 -26456.105} C_VEL
LIN {X 0,Y 104.288,Z 592.343,A -85,B 0,C 180,E1 -26460,E2 -26460} C_VEL
LIN {X 0,Y 106.036,Z 591.206,A -85,B 0,C 180,E1 -26466.137,E2 -26466.137} C_VEL
LIN {X 0,Y 114.842,Z 587.228,A -85,B 0,C 180,E1 -26477.818,E2 -26477.818} C_VEL
LIN {X 0,Y 122.604,Z 583.756,A -85,B 0,C 180,E1 -26483.476,E2 -26483.476} C_VEL
LIN {X 0,Y 125.409,Z 582.272,A -85,B 0,C 180,E1 -26484.854,E2 -26484.854} C_VEL
LIN {X 0,Y 132.749,Z 578.736,A -85,B 0,C 180,E1 -26488.456,E2 -26488.456} C_VEL
LIN {X 0,Y 138.728,Z 575.039,A -85,B 0,C 180,E1 -26490.438,E2 -26490.438} C_VEL
LIN {X 0,Y 141.407,Z 573.68,A -85,B 0,C 180,E1 -26491.457,E2 -26491.457} C_VEL
LIN {X 0,Y 147.424,Z 569.729,A -85,B 0,C 180,E1 -26493.127,E2 -26493.127} C_VEL
LIN {X 0,Y 148.829,Z 568.691,A -85,B 0,C 180,E1 -26493.458,E2 -26493.458} C_VEL
LIN {X 0,Y 148.53,Z 570.408,A -85,B 0,C 180,E1 -26494.096,E2 -26494.096} C_VEL
LIN {X 0,Y 142.219,Z 581.653,A -85,B 0,C 180,E1 -26496.513,E2 -26496.513} C_VEL
LIN {X 0,Y 136.027,Z 591.178,A -85,B 0,C 180,E1 -26499.19,E2 -26499.19} C_VEL
LIN {X 0,Y 128.913,Z 600.643,A -85,B 0,C 180,E1 -26502.604,E2 -26502.604} C_VEL
LIN {X 0,Y 121.364,Z 609.667,A -85,B 0,C 180,E1 -26507.118,E2 -26507.118} C_VEL
LIN {X 0,Y 114.6,Z 616.944,A -85,B 0,C 180,E1 -26512.169,E2 -26512.169} C_VEL
LIN {X 0,Y 109.709,Z 622.041,A -85,B 0,C 180,E1 -26517.003,E2 -26517.003} C_VEL
LIN {X 0,Y 104.422,Z 627.315,A -85,B 0,C 180,E1 -26524.052,E2 -26524.052} C_VEL
LIN {X 0,Y 101.349,Z 630.261,A -85,B 0,C 180,E1 -26529.708,E2 -26529.708} C_VEL
LIN {X 0,Y 98.882,Z 632.968,A -85,B 0,C 180,E1 -26537.684,E2 -26537.684} C_VEL
LIN {X 0,Y 97.952,Z 634.321,A -85,B 0,C 180,E1 -26545.88,E2 -26545.88} C_VEL
LIN {X 0,Y 97.947,Z 634.499,A -85,B 0,C 180,E1 -26549.995,E2 -26549.995} C_VEL
LIN {X 0,Y 98.248,Z 633.86,A -85,B 0,C 180,E1 -26558.22,E2 -26558.22} C_VEL
LIN {X 0,Y 99.881,Z 631.88,A -85,B 0,C 180,E1 -26566.342,E2 -26566.342} C_VEL
LIN {X 0,Y 103.232,Z 628.512,A -85,B 0,C 180,E1 -26574.104,E2 -26574.104} C_VEL
LIN {X 0,Y 108.233,Z 623.654,A -85,B 0,C 180,E1 -26581.291,E2 -26581.291} C_VEL
LIN {X 0,Y 114.568,Z 617.164,A -85,B 0,C 180,E1 -26587.832,E2 -26587.832} C_VEL
LIN {X 0,Y 121.275,Z 609.938,A -85,B 0,C 180,E1 -26592.91,E2 -26592.91} C_VEL
LIN {X 0,Y 128.815,Z 600.998,A -85,B 0,C 180,E1 -26597.432,E2 -26597.432} C_VEL
LIN {X 0,Y 135.895,Z 591.607,A -85,B 0,C 180,E1 -26600.866,E2 -26600.866} C_VEL
LIN {X 0,Y 142.892,Z 580.872,A -85,B 0,C 180,E1 -26603.828,E2 -26603.828} C_VEL
LIN {X 0,Y 149.147,Z 569.737,A -85,B 0,C 180,E1 -26606.145,E2 -26606.145} C_VEL
LIN {X 0,Y 155.195,Z 557.017,A -85,B 0,C 180,E1 -26608.106,E2 -26608.106} C_VEL
LIN {X 0,Y 159.985,Z 544.62,A -85,B 0,C 180,E1 -26609.547,E2 -26609.547} C_VEL
LIN {X 0,Y 164.161,Z 530.953,A -85,B 0,C 180,E1 -26610.696,E2 -26610.696} C_VEL
LIN {X 0,Y 167.19,Z 517.662,A -85,B 0,C 180,E1 -26611.448,E2 -26611.448} C_VEL
LIN {X 0,Y 169.241,Z 503.443,A -85,B 0,C 180,E1 -26611.995,E2 -26611.995} C_VEL
LIN {X 0,Y 172.05,Z 473.28,A -85,B 0,C 180,E1 -26612.889,E2 -26612.889} C_VEL
LIN {X 0,Y 170.451,Z 468.849,A -85,B 0,C 180,E1 -26614.377,E2 -26614.377} C_VEL
LIN {X 0,Y 166.932,Z 461.676,A -85,B 0,C 180,E1 -26617.806,E2 -26617.806} C_VEL
LIN {X 0,Y 164.019,Z 456.118,A -85,B 0,C 180,E1 -26621.173,E2 -26621.173} C_VEL
LIN {X 0,Y 161.975,Z 452.666,A -85,B 0,C 180,E1 -26623.954,E2 -26623.954} C_VEL
LIN {X 0,Y 160.5,Z 449.977,A -85,B 0,C 180,E1 -26626.387,E2 -26626.387} C_VEL
LIN {X 0,Y 158.69,Z 446.52,A -85,B 0,C 180,E1 -26630.279,E2 -26630.279} C_VEL
LIN {X 0,Y 156.931,Z 442.2,A -85,B 0,C 180,E1 -26640,E2 -26640} C_VEL
LIN {X 0,Y 158.904,Z 446.943,A -85,B 0,C 180,E1 -26650.31,E2 -26650.31} C_VEL
LIN {X 0,Y 161.332,Z 451.418,A -85,B 0,C 180,E1 -26655.071,E2 -26655.071} C_VEL
LIN {X 0,Y 163.608,Z 455.403,A -85,B 0,C 180,E1 -26658.348,E2 -26658.348} C_VEL
LIN {X 0,Y 166.426,Z 460.657,A -85,B 0,C 180,E1 -26661.692,E2 -26661.692} C_VEL
LIN {X 0,Y 170.164,Z 468.169,A -85,B 0,C 180,E1 -26665.401,E2 -26665.401} C_VEL
LIN {X 0,Y 172.066,Z 473.309,A -85,B 0,C 180,E1 -26667.169,E2 -26667.169} C_VEL
LIN {X 0,Y 168.332,Z 510.631,A -85,B 0,C 180,E1 -26668.281,E2 -26668.281} C_VEL
LIN {X 0,Y 165.643,Z 525.178,A -85,B 0,C 180,E1 -26669.014,E2 -26669.014} C_VEL
LIN {X 0,Y 161.8,Z 539.201,A -85,B 0,C 180,E1 -26670.009,E2 -26670.009} C_VEL
LIN {X 0,Y 157.262,Z 551.932,A -85,B 0,C 180,E1 -26671.281,E2 -26671.281} C_VEL
LIN {X 0,Y 151.851,Z 564.337,A -85,B 0,C 180,E1 -26672.987,E2 -26672.987} C_VEL
LIN {X 0,Y 145.931,Z 575.673,A -85,B 0,C 180,E1 -26675.051,E2 -26675.051} C_VEL
LIN {X 0,Y 139.648,Z 586.096,A -85,B 0,C 180,E1 -26677.574,E2 -26677.574} C_VEL
LIN {X 0,Y 132.381,Z 596.466,A -85,B 0,C 180,E1 -26680.848,E2 -26680.848} C_VEL
LIN {X 0,Y 125.572,Z 605.019,A -85,B 0,C 180,E1 -26684.478,E2 -26684.478} C_VEL
LIN {X 0,Y 118.313,Z 613.202,A -85,B 0,C 180,E1 -26689.206,E2 -26689.206} C_VEL
LIN {X 0,Y 111.705,Z 620.119,A -85,B 0,C 180,E1 -26694.875,E2 -26694.875} C_VEL
LIN {X 0,Y 106.882,Z 625.009,A -85,B 0,C 180,E1 -26700.457,E2 -26700.457} C_VEL
LIN {X 0,Y 103.24,Z 628.489,A -85,B 0,C 180,E1 -26705.898,E2 -26705.898} C_VEL
LIN {X 0,Y 99.882,Z 631.864,A -85,B 0,C 180,E1 -26713.659,E2 -26713.659} C_VEL
LIN {X 0,Y 98.247,Z 633.852,A -85,B 0,C 180,E1 -26721.78,E2 -26721.78} C_VEL
LIN {X 0,Y 97.946,Z 634.5,A -85,B 0,C 180,E1 -26730.005,E2 -26730.005} C_VEL
LIN {X 0,Y 98.295,Z 633.82,A -85,B 0,C 180,E1 -26738.227,E2 -26738.227} C_VEL
LIN {X 0,Y 99.079,Z 632.954,A -85,B 0,C 180,E1 -26742.382,E2 -26742.382} C_VEL
LIN {X 0,Y 99.391,Z 632.034,A -85,B 0,C 180,E1 -26745.741,E2 -26745.741} C_VEL
LIN {X 0,Y 98.845,Z 630.06,A -85,B 0,C 180,E1 -26751.367,E2 -26751.367} C_VEL
LIN {X 0,Y 99.326,Z 627.573,A -85,B 0,C 180,E1 -26756.9,E2 -26756.9} C_VEL
LIN {X 0,Y 101.163,Z 625.708,A -85,B 0,C 180,E1 -26759.919,E2 -26759.919} C_VEL
LIN {X 0,Y 107.946,Z 620.482,A -85,B 0,C 180,E1 -26765.876,E2 -26765.876} C_VEL
LIN {X 0,Y 109.614,Z 619.57,A -85,B 0,C 180,E1 -26766.953,E2 -26766.953} C_VEL
LIN {X 0,Y 118.008,Z 624.395,A -85,B 0,C 180,E1 -26773.232,E2 -26773.232} C_VEL
LIN {X 0,Y 120.237,Z 625.408,A -85,B 0,C 180,E1 -26774.546,E2 -26774.546} C_VEL
LIN {X 0,Y 121.169,Z 625.766,A -85,B 0,C 180,E1 -26775.892,E2 -26775.892} C_VEL
LIN {X 0,Y 112.719,Z 621.482,A -85,B 0,C 180,E1 -26781.428,E2 -26781.428} C_VEL
LIN {X 0,Y 105.986,Z 616.169,A -85,B 0,C 180,E1 -26787.962,E2 -26787.962} C_VEL
LIN {X 0,Y 101.187,Z 609.655,A -85,B 0,C 180,E1 -26795.372,E2 -26795.372} C_VEL
LIN {X 0,Y 98.369,Z 601.537,A -85,B 0,C 180,E1 -26803.928,E2 -26803.928} C_VEL
LIN {X 0,Y 97.803,Z 600.922,A -85,B 0,C 180,E1 -26805.434,E2 -26805.434} C_VEL
LIN {X 0,Y 97.269,Z 600.607,A -85,B 0,C 180,E1 -26807.482,E2 -26807.482} C_VEL
LIN {X 0,Y 98.195,Z 598.102,A -85,B 0,C 180,E1 -26815.896,E2 -26815.896} C_VEL
LIN {X 0,Y 98.955,Z 597.233,A -85,B 0,C 180,E1 -26820,E2 -26820} C_VEL
LIN {X 0,Y 99.875,Z 596.651,A -85,B 0,C 180,E1 -26824.035,E2 -26824.035} C_VEL
LIN {X 0,Y 106.699,Z 593.592,A -85,B 0,C 180,E1 -26835.276,E2 -26835.276} C_VEL
LIN {X 0,Y 113.765,Z 590.956,A -85,B 0,C 180,E1 -26841.757,E2 -26841.757} C_VEL
LIN {X 0,Y 120.563,Z 588.148,A -85,B 0,C 180,E1 -26845.926,E2 -26845.926} C_VEL
LIN {X 0,Y 130.342,Z 583.76,A -85,B 0,C 180,E1 -26850.371,E2 -26850.371} C_VEL
LIN {X 0,Y 138.004,Z 579.537,A -85,B 0,C 180,E1 -26852.765,E2 -26852.765} C_VEL
LIN {X 0,Y 139.044,Z 579.063,A -85,B 0,C 180,E1 -26853.132,E2 -26853.132} C_VEL
LIN {X 0,Y 138.957,Z 580.244,A -85,B 0,C 180,E1 -26853.804,E2 -26853.804} C_VEL
LIN {X 0,Y 131.655,Z 591.181,A -85,B 0,C 180,E1 -26856.795,E2 -26856.795} C_VEL
LIN {X 0,Y 124.205,Z 600.646,A -85,B 0,C 180,E1 -26860.187,E2 -26860.187} C_VEL
LIN {X 0,Y 116.24,Z 609.669,A -85,B 0,C 180,E1 -26864.725,E2 -26864.725} C_VEL
LIN {X 0,Y 109.072,Z 616.946,A -85,B 0,C 180,E1 -26869.878,E2 -26869.878} C_VEL
LIN {X 0,Y 103.677,Z 622.146,A -85,B 0,C 180,E1 -26874.969,E2 -26874.969} C_VEL
LIN {X 0,Y 98.047,Z 627.316,A -85,B 0,C 180,E1 -26882.225,E2 -26882.225} C_VEL
LIN {X 0,Y 94.682,Z 630.261,A -85,B 0,C 180,E1 -26888.209,E2 -26888.209} C_VEL
LIN {X 0,Y 91.924,Z 632.968,A -85,B 0,C 180,E1 -26896.735,E2 -26896.735} C_VEL
LIN {X 0,Y 90.882,Z 634.321,A -85,B 0,C 180,E1 -26905.559,E2 -26905.559} C_VEL
LIN {X 0,Y 90.846,Z 634.499,A -85,B 0,C 180,E1 -26909.994,E2 -26909.994} C_VEL
LIN {X 0,Y 90.88,Z 634.345,A -85,B 0,C 180,E1 -26914.43,E2 -26914.43} C_VEL
LIN {X 0,Y 91.886,Z 633.039,A -85,B 0,C 180,E1 -26923.259,E2 -26923.259} C_VEL
LIN {X 0,Y 94.662,Z 630.374,A -85,B 0,C 180,E1 -26931.784,E2 -26931.784} C_VEL
LIN {X 0,Y 99.327,Z 626.276,A -85,B 0,C 180,E1 -26939.683,E2 -26939.683} C_VEL
LIN {X 0,Y 105.415,Z 620.623,A -85,B 0,C 180,E1 -26946.866,E2 -26946.866} C_VEL
LIN {X 0,Y 111.954,Z 614.247,A -85,B 0,C 180,E1 -26952.435,E2 -26952.435} C_VEL
LIN {X 0,Y 119.491,Z 606.321,A -85,B 0,C 180,E1 -26957.317,E2 -26957.317} C_VEL
LIN {X 0,Y 126.535,Z 598.029,A -85,B 0,C 180,E1 -26961.033,E2 -26961.033} C_VEL
LIN {X 0,Y 134.07,Z 588.042,A -85,B 0,C 180,E1 -26964.335,E2 -26964.335} C_VEL
LIN {X 0,Y 141.212,Z 576.975,A -85,B 0,C 180,E1 -26967.084,E2 -26967.084} C_VEL
LIN {X 0,Y 147.383,Z 565.85,A -85,B 0,C 180,E1 -26969.122,E2 -26969.122} C_VEL
LIN {X 0,Y 152.979,Z 553.819,A -85,B 0,C 180,E1 -26970.787,E2 -26970.787} C_VEL
LIN {X 0,Y 157.953,Z 540.487,A -85,B 0,C 180,E1 -26972.161,E2 -26972.161} C_VEL
LIN {X 0,Y 161.877,Z 526.857,A -85,B 0,C 180,E1 -26973.155,E2 -26973.155} C_VEL
LIN {X 0,Y 164.859,Z 512.109,A -85,B 0,C 180,E1 -26973.874,E2 -26973.874} C_VEL
LIN {X 0,Y 167.235,Z 491.043,A -85,B 0,C 180,E1 -26974.515,E2 -26974.515} C_VEL
LIN {X 0,Y 168.634,Z 476.182,A -85,B 0,C 180,E1 -26974.962,E2 -26974.962} C_VEL
LIN {X 0,Y 166.73,Z 471.6,A -85,B 0,C 180,E1 -26976.887,E2 -26976.887} C_VEL
LIN {X 0,Y 163.361,Z 464.568,A -85,B 0,C 180,E1 -26980.728,E2 -26980.728} C_VEL
LIN {X 0,Y 161.137,Z 460.316,A -85,B 0,C 180,E1 -26983.783,E2 -26983.783} C_VEL
LIN {X 0,Y 159.193,Z 456.695,A -85,B 0,C 180,E1 -26987.085,E2 -26987.085} C_VEL
LIN {X 0,Y 157.508,Z 453.323,A -85,B 0,C 180,E1 -26991.015,E2 -26991.015} C_VEL
LIN {X 0,Y 156.061,Z 449.291,A -85,B 0,C 180,E1 -27000,E2 -27000} C_VEL
LIN {X 0,Y 157.726,Z 453.704,A -85,B 0,C 180,E1 -27009.619,E2 -27009.619} C_VEL
LIN {X 0,Y 159.886,Z 457.984,A -85,B 0,C 180,E1 -27014.234,E2 -27014.234} C_VEL
LIN {X 0,Y 162.012,Z 461.943,A -85,B 0,C 180,E1 -27017.53,E2 -27017.53} C_VEL
LIN {X 0,Y 164.587,Z 467.044,A -85,B 0,C 180,E1 -27020.802,E2 -27020.802} C_VEL
LIN {X 0,Y 167.893,Z 474.184,A -85,B 0,C 180,E1 -27024.334,E2 -27024.334} C_VEL
LIN {X 0,Y 168.643,Z 476.296,A -85,B 0,C 180,E1 -27025.101,E2 -27025.101} C_VEL
LIN {X 0,Y 165.122,Z 510.433,A -85,B 0,C 180,E1 -27026.102,E2 -27026.102} C_VEL
LIN {X 0,Y 162.439,Z 524.657,A -85,B 0,C 180,E1 -27026.786,E2 -27026.786} C_VEL
LIN {X 0,Y 158.37,Z 539.208,A -85,B 0,C 180,E1 -27027.785,E2 -27027.785} C_VEL
LIN {X 0,Y 153.699,Z 551.938,A -85,B 0,C 180,E1 -27029.021,E2 -27029.021} C_VEL
LIN {X 0,Y 148.103,Z 564.341,A -85,B 0,C 180,E1 -27030.681,E2 -27030.681} C_VEL
LIN {X 0,Y 141.96,Z 575.676,A -85,B 0,C 180,E1 -27032.696,E2 -27032.696} C_VEL
LIN {X 0,Y 135.422,Z 586.099,A -85,B 0,C 180,E1 -27035.184,E2 -27035.184} C_VEL
LIN {X 0,Y 127.847,Z 596.468,A -85,B 0,C 180,E1 -27038.439,E2 -27038.439} C_VEL
LIN {X 0,Y 120.685,Z 605.022,A -85,B 0,C 180,E1 -27042.063,E2 -27042.063} C_VEL
LIN {X 0,Y 113.025,Z 613.203,A -85,B 0,C 180,E1 -27046.85,E2 -27046.85} C_VEL
LIN {X 0,Y 105.52,Z 620.511,A -85,B 0,C 180,E1 -27053.057,E2 -27053.057} C_VEL
LIN {X 0,Y 99.361,Z 626.252,A -85,B 0,C 180,E1 -27060.328,E2 -27060.328} C_VEL
LIN {X 0,Y 94.667,Z 630.356,A -85,B 0,C 180,E1 -27068.217,E2 -27068.217} C_VEL
LIN {X 0,Y 91.907,Z 633.028,A -85,B 0,C 180,E1 -27076.744,E2 -27076.744} C_VEL
LIN {X 0,Y 90.879,Z 634.342,A -85,B 0,C 180,E1 -27085.57,E2 -27085.57} C_VEL
LIN {X 0,Y 90.845,Z 634.5,A -85,B 0,C 180,E1 -27090.006,E2 -27090.006} C_VEL
LIN {X 0,Y 91.266,Z 633.819,A -85,B 0,C 180,E1 -27098.865,E2 -27098.865} C_VEL
LIN {X 0,Y 93.489,Z 631.802,A -85,B 0,C 180,E1 -27107.505,E2 -27107.505} C_VEL
LIN {X 0,Y 97.741,Z 628.4,A -85,B 0,C 180,E1 -27115.564,E2 -27115.564} C_VEL
LIN {X 0,Y 101.163,Z 625.708,A -85,B 0,C 180,E1 -27119.919,E2 -27119.919} C_VEL
LIN {X 0,Y 102.414,Z 624.475,A -85,B 0,C 180,E1 -27121.895,E2 -27121.895} C_VEL
LIN {X 0,Y 103.217,Z 622.112,A -85,B 0,C 180,E1 -27125.306,E2 -27125.306} C_VEL
LIN {X 0,Y 104.347,Z 619.547,A -85,B 0,C 180,E1 -27128.706,E2 -27128.706} C_VEL
LIN {X 0,Y 105.941,Z 618.144,A -85,B 0,C 180,E1 -27130.449,E2 -27130.449} C_VEL
LIN {X 0,Y 106.142,Z 618.167,A -85,B 0,C 180,E1 -27130.6,E2 -27130.6} C_VEL
LIN {X 0,Y 112.07,Z 621.6,A -85,B 0,C 180,E1 -27134.87,E2 -27134.87} C_VEL
LIN {X 0,Y 111.838,Z 621.462,A -85,B 0,C 180,E1 -27136.271,E2 -27136.271} C_VEL
LIN {X 0,Y 103.835,Z 616.256,A -85,B 0,C 180,E1 -27142.472,E2 -27142.472} C_VEL
LIN {X 0,Y 96.432,Z 608.552,A -85,B 0,C 180,E1 -27151.723,E2 -27151.723} C_VEL
LIN {X 0,Y 94.952,Z 608.038,A -85,B 0,C 180,E1 -27153.635,E2 -27153.635} C_VEL
LIN {X 0,Y 92.944,Z 607.341,A -85,B 0,C 180,E1 -27157.786,E2 -27157.786} C_VEL
LIN {X 0,Y 92.396,Z 605.967,A -85,B 0,C 180,E1 -27162.287,E2 -27162.287} C_VEL
LIN {X 0,Y 92.526,Z 602.746,A -85,B 0,C 180,E1 -27175.644,E2 -27175.644} C_VEL
LIN {X 0,Y 93.391,Z 601.864,A -85,B 0,C 180,E1 -27180,E2 -27180} C_VEL
LIN {X 0,Y 96.159,Z 600.465,A -85,B 0,C 180,E1 -27188.406,E2 -27188.406} C_VEL
LIN {X 0,Y 104.856,Z 597.359,A -85,B 0,C 180,E1 -27199.581,E2 -27199.581} C_VEL
LIN {X 0,Y 113.263,Z 594.425,A -85,B 0,C 180,E1 -27205.744,E2 -27205.744} C_VEL
LIN {X 0,Y 125.774,Z 589.463,A -85,B 0,C 180,E1 -27211.598,E2 -27211.598} C_VEL
LIN {X 0,Y 129.409,Z 587.907,A -85,B 0,C 180,E1 -27212.894,E2 -27212.894} C_VEL
LIN {X 0,Y 129.211,Z 588.903,A -85,B 0,C 180,E1 -27213.556,E2 -27213.556} C_VEL
LIN {X 0,Y 120.992,Z 599.163,A -85,B 0,C 180,E1 -27216.989,E2 -27216.989} C_VEL
LIN {X 0,Y 113.663,Z 607.259,A -85,B 0,C 180,E1 -27220.754,E2 -27220.754} C_VEL
LIN {X 0,Y 105.827,Z 615.015,A -85,B 0,C 180,E1 -27225.782,E2 -27225.782} C_VEL
LIN {X 0,Y 98.331,Z 621.731,A -85,B 0,C 180,E1 -27232.081,E2 -27232.081} C_VEL
LIN {X 0,Y 93.237,Z 626.127,A -85,B 0,C 180,E1 -27238.147,E2 -27238.147} C_VEL
LIN {X 0,Y 88.093,Z 630.262,A -85,B 0,C 180,E1 -27246.485,E2 -27246.485} C_VEL
LIN {X 0,Y 85.006,Z 632.969,A -85,B 0,C 180,E1 -27255.633,E2 -27255.633} C_VEL
LIN {X 0,Y 83.8,Z 634.322,A -85,B 0,C 180,E1 -27265.183,E2 -27265.183} C_VEL
LIN {X 0,Y 83.768,Z 634.499,A -85,B 0,C 180,E1 -27269.994,E2 -27269.994} C_VEL
LIN {X 0,Y 83.797,Z 634.345,A -85,B 0,C 180,E1 -27274.805,E2 -27274.805} C_VEL
LIN {X 0,Y 84.974,Z 633.039,A -85,B 0,C 180,E1 -27284.36,E2 -27284.36} C_VEL
LIN {X 0,Y 88.072,Z 630.373,A -85,B 0,C 180,E1 -27293.509,E2 -27293.509} C_VEL
LIN {X 0,Y 93.174,Z 626.275,A -85,B 0,C 180,E1 -27301.864,E2 -27301.864} C_VEL
LIN {X 0,Y 99.79,Z 620.622,A -85,B 0,C 180,E1 -27309.328,E2 -27309.328} C_VEL
LIN {X 0,Y 106.809,Z 614.246,A -85,B 0,C 180,E1 -27315.012,E2 -27315.012} C_VEL
LIN {X 0,Y 114.774,Z 606.319,A -85,B 0,C 180,E1 -27319.937,E2 -27319.937} C_VEL
LIN {X 0,Y 122.187,Z 598.027,A -85,B 0,C 180,E1 -27323.627,E2 -27323.627} C_VEL
LIN {X 0,Y 130.039,Z 588.039,A -85,B 0,C 180,E1 -27326.891,E2 -27326.891} C_VEL
LIN {X 0,Y 137.508,Z 576.917,A -85,B 0,C 180,E1 -27329.587,E2 -27329.587} C_VEL
LIN {X 0,Y 143.872,Z 565.845,A -85,B 0,C 180,E1 -27331.548,E2 -27331.548} C_VEL
LIN {X 0,Y 149.639,Z 553.813,A -85,B 0,C 180,E1 -27333.163,E2 -27333.163} C_VEL
LIN {X 0,Y 154.766,Z 540.48,A -85,B 0,C 180,E1 -27334.484,E2 -27334.484} C_VEL
LIN {X 0,Y 158.73,Z 527.112,A -85,B 0,C 180,E1 -27335.429,E2 -27335.429} C_VEL
LIN {X 0,Y 161.745,Z 512.85,A -85,B 0,C 180,E1 -27336.094,E2 -27336.094} C_VEL
LIN {X 0,Y 163.989,Z 494.159,A -85,B 0,C 180,E1 -27336.667,E2 -27336.667} C_VEL
LIN {X 0,Y 165.419,Z 479.463,A -85,B 0,C 180,E1 -27337.1,E2 -27337.1} C_VEL
LIN {X 0,Y 162.223,Z 472.195,A -85,B 0,C 180,E1 -27340.875,E2 -27340.875} C_VEL
LIN {X 0,Y 159.852,Z 467.19,A -85,B 0,C 180,E1 -27344.29,E2 -27344.29} C_VEL
LIN {X 0,Y 157.871,Z 463.347,A -85,B 0,C 180,E1 -27347.873,E2 -27347.873} C_VEL
LIN {X 0,Y 156.408,Z 460.196,A -85,B 0,C 180,E1 -27351.602,E2 -27351.602} C_VEL
LIN {X 0,Y 155.187,Z 456.407,A -85,B 0,C 180,E1 -27360,E2 -27360} C_VEL
LIN {X 0,Y 156.652,Z 460.678,A -85,B 0,C 180,E1 -27369.164,E2 -27369.164} C_VEL
LIN {X 0,Y 158.497,Z 464.586,A -85,B 0,C 180,E1 -27373.421,E2 -27373.421} C_VEL
LIN {X 0,Y 160.709,Z 468.972,A -85,B 0,C 180,E1 -27377.074,E2 -27377.074} C_VEL
LIN {X 0,Y 163.815,Z 475.708,A -85,B 0,C 180,E1 -27381.137,E2 -27381.137} C_VEL
LIN {X 0,Y 165.458,Z 479.603,A -85,B 0,C 180,E1 -27382.992,E2 -27382.992} C_VEL
LIN {X 0,Y 162.13,Z 510.443,A -85,B 0,C 180,E1 -27383.853,E2 -27383.853} C_VEL
LIN {X 0,Y 159.433,Z 524.406,A -85,B 0,C 180,E1 -27384.494,E2 -27384.494} C_VEL
LIN {X 0,Y 155.556,Z 538.086,A -85,B 0,C 180,E1 -27385.374,E2 -27385.374} C_VEL
LIN {X 0,Y 150.384,Z 551.943,A -85,B 0,C 180,E1 -27386.656,E2 -27386.656} C_VEL
LIN {X 0,Y 144.615,Z 564.346,A -85,B 0,C 180,E1 -27388.265,E2 -27388.265} C_VEL
LIN {X 0,Y 137.605,Z 576.77,A -85,B 0,C 180,E1 -27390.433,E2 -27390.433} C_VEL
LIN {X 0,Y 130.134,Z 587.983,A -85,B 0,C 180,E1 -27393.174,E2 -27393.174} C_VEL
LIN {X 0,Y 122.241,Z 597.979,A -85,B 0,C 180,E1 -27396.407,E2 -27396.407} C_VEL
LIN {X 0,Y 114.839,Z 606.278,A -85,B 0,C 180,E1 -27400.102,E2 -27400.102} C_VEL
LIN {X 0,Y 106.826,Z 614.212,A -85,B 0,C 180,E1 -27404.997,E2 -27404.997} C_VEL
LIN {X 0,Y 99.494,Z 620.875,A -85,B 0,C 180,E1 -27410.988,E2 -27410.988} C_VEL
LIN {X 0,Y 93.217,Z 626.253,A -85,B 0,C 180,E1 -27418.153,E2 -27418.153} C_VEL
LIN {X 0,Y 88.077,Z 630.357,A -85,B 0,C 180,E1 -27426.493,E2 -27426.493} C_VEL
LIN {X 0,Y 84.991,Z 633.029,A -85,B 0,C 180,E1 -27435.643,E2 -27435.643} C_VEL
LIN {X 0,Y 83.796,Z 634.342,A -85,B 0,C 180,E1 -27445.195,E2 -27445.195} C_VEL
LIN {X 0,Y 83.767,Z 634.5,A -85,B 0,C 180,E1 -27450.006,E2 -27450.006} C_VEL
LIN {X 0,Y 84.245,Z 633.819,A -85,B 0,C 180,E1 -27459.611,E2 -27459.611} C_VEL
LIN {X 0,Y 86.742,Z 631.801,A -85,B 0,C 180,E1 -27468.916,E2 -27468.916} C_VEL
LIN {X 0,Y 91.379,Z 628.399,A -85,B 0,C 180,E1 -27477.487,E2 -27477.487} C_VEL
LIN {X 0,Y 96.255,Z 624.909,A -85,B 0,C 180,E1 -27483.209,E2 -27483.209} C_VEL
LIN {X 0,Y 102.285,Z 620.461,A -85,B 0,C 180,E1 -27488.204,E2 -27488.204} C_VEL
LIN {X 0,Y 105.932,Z 618.123,A -85,B 0,C 180,E1 -27490.467,E2 -27490.467} C_VEL
LIN {X 0,Y 106.142,Z 618.167,A -85,B 0,C 180,E1 -27490.6,E2 -27490.6} C_VEL
LIN {X 0,Y 106.905,Z 618.665,A -85,B 0,C 180,E1 -27491.79,E2 -27491.79} C_VEL
LIN {X 0,Y 106.561,Z 618.58,A -85,B 0,C 180,E1 -27493.435,E2 -27493.435} C_VEL
LIN {X 0,Y 105.031,Z 617.684,A -85,B 0,C 180,E1 -27495.343,E2 -27495.343} C_VEL
LIN {X 0,Y 100.993,Z 615.368,A -85,B 0,C 180,E1 -27498.361,E2 -27498.361} C_VEL
LIN {X 0,Y 98.133,Z 614.126,A -85,B 0,C 180,E1 -27500.482,E2 -27500.482} C_VEL
LIN {X 0,Y 97.217,Z 613.947,A -85,B 0,C 180,E1 -27501.249,E2 -27501.249} C_VEL
LIN {X 0,Y 94.7,Z 613.668,A -85,B 0,C 180,E1 -27503.58,E2 -27503.58} C_VEL
LIN {X 0,Y 89.641,Z 611.916,A -85,B 0,C 180,E1 -27511.939,E2 -27511.939} C_VEL
LIN {X 0,Y 87.424,Z 611.316,A -85,B 0,C 180,E1 -27516.3,E2 -27516.3} C_VEL
LIN {X 0,Y 85.976,Z 608.188,A -85,B 0,C 180,E1 -27530.591,E2 -27530.591} C_VEL
LIN {X 0,Y 87.624,Z 606.213,A -85,B 0,C 180,E1 -27540,E2 -27540} C_VEL
LIN {X 0,Y 90.546,Z 604.897,A -85,B 0,C 180,E1 -27548.931,E2 -27548.931} C_VEL
LIN {X 0,Y 99.575,Z 602.025,A -85,B 0,C 180,E1 -27560.665,E2 -27560.665} C_VEL
LIN {X 0,Y 108.237,Z 599.368,A -85,B 0,C 180,E1 -27567.035,E2 -27567.035} C_VEL
LIN {X 0,Y 116.583,Z 596.533,A -85,B 0,C 180,E1 -27571.184,E2 -27571.184} C_VEL
LIN {X 0,Y 118.932,Z 595.627,A -85,B 0,C 180,E1 -27572.13,E2 -27572.13} C_VEL
LIN {X 0,Y 119.405,Z 596.318,A -85,B 0,C 180,E1 -27573.15,E2 -27573.15} C_VEL
LIN {X 0,Y 111.645,Z 604.753,A -85,B 0,C 180,E1 -27576.613,E2 -27576.613} C_VEL
LIN {X 0,Y 103.122,Z 613,A -85,B 0,C 180,E1 -27581.431,E2 -27581.431} C_VEL
LIN {X 0,Y 96.452,Z 618.758,A -85,B 0,C 180,E1 -27586.187,E2 -27586.187} C_VEL
LIN {X 0,Y 90.628,Z 623.486,A -85,B 0,C 180,E1 -27591.649,E2 -27591.649} C_VEL
LIN {X 0,Y 84.207,Z 628.381,A -85,B 0,C 180,E1 -27599.943,E2 -27599.943} C_VEL
LIN {X 0,Y 79.596,Z 631.789,A -85,B 0,C 180,E1 -27609.311,E2 -27609.311} C_VEL
LIN {X 0,Y 77.201,Z 633.812,A -85,B 0,C 180,E1 -27619.503,E2 -27619.503} C_VEL
LIN {X 0,Y 76.739,Z 634.322,A -85,B 0,C 180,E1 -27624.739,E2 -27624.739} C_VEL
LIN {X 0,Y 76.68,Z 634.499,A -85,B 0,C 180,E1 -27629.993,E2 -27629.993} C_VEL
LIN {X 0,Y 76.734,Z 634.345,A -85,B 0,C 180,E1 -27635.248,E2 -27635.248} C_VEL
LIN {X 0,Y 78.079,Z 633.038,A -85,B 0,C 180,E1 -27645.659,E2 -27645.659} C_VEL
LIN {X 0,Y 81.576,Z 630.372,A -85,B 0,C 180,E1 -27655.509,E2 -27655.509} C_VEL
LIN {X 0,Y 87.178,Z 626.274,A -85,B 0,C 180,E1 -27664.347,E2 -27664.347} C_VEL
LIN {X 0,Y 93.383,Z 621.424,A -85,B 0,C 180,E1 -27671.184,E2 -27671.184} C_VEL
LIN {X 0,Y 100.741,Z 615.251,A -85,B 0,C 180,E1 -27677.089,E2 -27677.089} C_VEL
LIN {X 0,Y 109.077,Z 607.548,A -85,B 0,C 180,E1 -27682.111,E2 -27682.111} C_VEL
LIN {X 0,Y 116.771,Z 599.509,A -85,B 0,C 180,E1 -27685.84,E2 -27685.84} C_VEL
LIN {X 0,Y 124.847,Z 589.909,A -85,B 0,C 180,E1 -27689.056,E2 -27689.056} C_VEL
LIN {X 0,Y 132.415,Z 579.381,A -85,B 0,C 180,E1 -27691.68,E2 -27691.68} C_VEL
LIN {X 0,Y 139.139,Z 568.433,A -85,B 0,C 180,E1 -27693.7,E2 -27693.7} C_VEL
LIN {X 0,Y 145.074,Z 557.002,A -85,B 0,C 180,E1 -27695.266,E2 -27695.266} C_VEL
LIN {X 0,Y 150.318,Z 544.601,A -85,B 0,C 180,E1 -27696.561,E2 -27696.561} C_VEL
LIN {X 0,Y 154.744,Z 531.352,A -85,B 0,C 180,E1 -27697.545,E2 -27697.545} C_VEL
LIN {X 0,Y 158.167,Z 517.407,A -85,B 0,C 180,E1 -27698.254,E2 -27698.254} C_VEL
LIN {X 0,Y 160.373,Z 503.224,A -85,B 0,C 180,E1 -27698.729,E2 -27698.729} C_VEL
LIN {X 0,Y 162.439,Z 483.259,A -85,B 0,C 180,E1 -27699.26,E2 -27699.26} C_VEL
LIN {X 0,Y 159.428,Z 476.043,A -85,B 0,C 180,E1 -27703.414,E2 -27703.414} C_VEL
LIN {X 0,Y 157.649,Z 472.331,A -85,B 0,C 180,E1 -27706.428,E2 -27706.428} C_VEL
LIN {X 0,Y 156.443,Z 469.709,A -85,B 0,C 180,E1 -27708.993,E2 -27708.993} C_VEL
LIN {X 0,Y 155.254,Z 466.917,A -85,B 0,C 180,E1 -27712.44,E2 -27712.44} C_VEL
LIN {X 0,Y 154.312,Z 463.532,A -85,B 0,C 180,E1 -27720,E2 -27720} C_VEL
LIN {X 0,Y 155.573,Z 467.594,A -85,B 0,C 180,E1 -27728.647,E2 -27728.647} C_VEL
LIN {X 0,Y 157.214,Z 471.363,A -85,B 0,C 180,E1 -27732.751,E2 -27732.751} C_VEL
LIN {X 0,Y 159.11,Z 475.411,A -85,B 0,C 180,E1 -27736.143,E2 -27736.143} C_VEL
LIN {X 0,Y 161.814,Z 481.744,A -85,B 0,C 180,E1 -27740.001,E2 -27740.001} C_VEL
LIN {X 0,Y 162.446,Z 483.321,A -85,B 0,C 180,E1 -27740.799,E2 -27740.799} C_VEL
LIN {X 0,Y 159.49,Z 509.905,A -85,B 0,C 180,E1 -27741.504,E2 -27741.504} C_VEL
LIN {X 0,Y 156.73,Z 524.016,A -85,B 0,C 180,E1 -27742.115,E2 -27742.115} C_VEL
LIN {X 0,Y 152.647,Z 538.093,A -85,B 0,C 180,E1 -27742.964,E2 -27742.964} C_VEL
LIN {X 0,Y 147.333,Z 551.949,A -85,B 0,C 180,E1 -27744.186,E2 -27744.186} C_VEL
LIN {X 0,Y 141.395,Z 564.35,A -85,B 0,C 180,E1 -27745.733,E2 -27745.733} C_VEL
LIN {X 0,Y 134.81,Z 575.684,A -85,B 0,C 180,E1 -27747.602,E2 -27747.602} C_VEL
LIN {X 0,Y 127.744,Z 586.106,A -85,B 0,C 180,E1 -27749.953,E2 -27749.953} C_VEL
LIN {X 0,Y 119.523,Z 596.473,A -85,B 0,C 180,E1 -27753.089,E2 -27753.089} C_VEL
LIN {X 0,Y 111.614,Z 605.026,A -85,B 0,C 180,E1 -27756.607,E2 -27756.607} C_VEL
LIN {X 0,Y 103.085,Z 613.207,A -85,B 0,C 180,E1 -27761.423,E2 -27761.423} C_VEL
LIN {X 0,Y 96.446,Z 618.939,A -85,B 0,C 180,E1 -27766.199,E2 -27766.199} C_VEL
LIN {X 0,Y 90.658,Z 623.628,A -85,B 0,C 180,E1 -27771.679,E2 -27771.679} C_VEL
LIN {X 0,Y 84.189,Z 628.492,A -85,B 0,C 180,E1 -27779.949,E2 -27779.949} C_VEL
LIN {X 0,Y 79.585,Z 631.866,A -85,B 0,C 180,E1 -27789.322,E2 -27789.322} C_VEL
LIN {X 0,Y 77.181,Z 633.853,A -85,B 0,C 180,E1 -27799.514,E2 -27799.514} C_VEL
LIN {X 0,Y 76.734,Z 634.342,A -85,B 0,C 180,E1 -27804.752,E2 -27804.752} C_VEL
LIN {X 0,Y 76.679,Z 634.5,A -85,B 0,C 180,E1 -27810.007,E2 -27810.007} C_VEL
LIN {X 0,Y 77.254,Z 633.819,A -85,B 0,C 180,E1 -27820.49,E2 -27820.49} C_VEL
LIN {X 0,Y 80.063,Z 631.801,A -85,B 0,C 180,E1 -27830.563,E2 -27830.563} C_VEL
LIN {X 0,Y 85.135,Z 628.398,A -85,B 0,C 180,E1 -27839.696,E2 -27839.696} C_VEL
LIN {X 0,Y 90.394,Z 624.908,A -85,B 0,C 180,E1 -27845.677,E2 -27845.677} C_VEL
LIN {X 0,Y 96.816,Z 620.46,A -85,B 0,C 180,E1 -27850.799,E2 -27850.799} C_VEL
LIN {X 0,Y 102.872,Z 616.49,A -85,B 0,C 180,E1 -27854.283,E2 -27854.283} C_VEL
LIN {X 0,Y 104.107,Z 617.123,A -85,B 0,C 180,E1 -27855.146,E2 -27855.146} C_VEL
LIN {X 0,Y 103.759,Z 616.893,A -85,B 0,C 180,E1 -27856.089,E2 -27856.089} C_VEL
LIN {X 0,Y 99.648,Z 614.371,A -85,B 0,C 180,E1 -27859.279,E2 -27859.279} C_VEL
LIN {X 0,Y 97.217,Z 613.947,A -85,B 0,C 180,E1 -27861.249,E2 -27861.249} C_VEL
LIN {X 0,Y 92.42,Z 613.925,A -85,B 0,C 180,E1 -27865.058,E2 -27865.058} C_VEL
LIN {X 0,Y 83.207,Z 614.672,A -85,B 0,C 180,E1 -27873.469,E2 -27873.469} C_VEL
LIN {X 0,Y 81.134,Z 614.442,A -85,B 0,C 180,E1 -27877.289,E2 -27877.289} C_VEL
LIN {X 0,Y 80.76,Z 614.23,A -85,B 0,C 180,E1 -27878.638,E2 -27878.638} C_VEL
LIN {X 0,Y 81.622,Z 610.302,A -85,B 0,C 180,E1 -27900,E2 -27900} C_VEL
LIN {X 0,Y 87.358,Z 608.203,A -85,B 0,C 180,E1 -27913.967,E2 -27913.967} C_VEL
LIN {X 0,Y 98.372,Z 605.319,A -85,B 0,C 180,E1 -27925.383,E2 -27925.383} C_VEL
LIN {X 0,Y 108.305,Z 602.481,A -85,B 0,C 180,E1 -27931.274,E2 -27931.274} C_VEL
LIN {X 0,Y 109.862,Z 602.014,A -85,B 0,C 180,E1 -27931.995,E2 -27931.995} C_VEL
LIN {X 0,Y 108.877,Z 603.401,A -85,B 0,C 180,E1 -27932.942,E2 -27932.942} C_VEL
LIN {X 0,Y 99.784,Z 611.906,A -85,B 0,C 180,E1 -27937.586,E2 -27937.586} C_VEL
LIN {X 0,Y 91.442,Z 618.759,A -85,B 0,C 180,E1 -27943.093,E2 -27943.093} C_VEL
LIN {X 0,Y 85.139,Z 623.487,A -85,B 0,C 180,E1 -27948.664,E2 -27948.664} C_VEL
LIN {X 0,Y 78.113,Z 628.382,A -85,B 0,C 180,E1 -27957.321,E2 -27957.321} C_VEL
LIN {X 0,Y 72.963,Z 631.789,A -85,B 0,C 180,E1 -27967.331,E2 -27967.331} C_VEL
LIN {X 0,Y 70.211,Z 633.812,A -85,B 0,C 180,E1 -27978.444,E2 -27978.444} C_VEL
LIN {X 0,Y 69.655,Z 634.322,A -85,B 0,C 180,E1 -27984.202,E2 -27984.202} C_VEL
LIN {X 0,Y 69.582,Z 634.499,A -85,B 0,C 180,E1 -27989.993,E2 -27989.993} C_VEL
LIN {X 0,Y 69.647,Z 634.345,A -85,B 0,C 180,E1 -27995.784,E2 -27995.784} C_VEL
LIN {X 0,Y 71.243,Z 633.038,A -85,B 0,C 180,E1 -28007.206,E2 -28007.206} C_VEL
LIN {X 0,Y 75.196,Z 630.372,A -85,B 0,C 180,E1 -28017.852,E2 -28017.852} C_VEL
LIN {X 0,Y 81.374,Z 626.273,A -85,B 0,C 180,E1 -28027.189,E2 -28027.189} C_VEL
LIN {X 0,Y 89.205,Z 620.619,A -85,B 0,C 180,E1 -28035.15,E2 -28035.15} C_VEL
LIN {X 0,Y 97.25,Z 614.243,A -85,B 0,C 180,E1 -28040.966,E2 -28040.966} C_VEL
LIN {X 0,Y 106.143,Z 606.315,A -85,B 0,C 180,E1 -28045.85,E2 -28045.85} C_VEL
LIN {X 0,Y 114.326,Z 598.022,A -85,B 0,C 180,E1 -28049.378,E2 -28049.378} C_VEL
LIN {X 0,Y 123.429,Z 587.29,A -85,B 0,C 180,E1 -28052.669,E2 -28052.669} C_VEL
LIN {X 0,Y 131.618,Z 575.745,A -85,B 0,C 180,E1 -28055.186,E2 -28055.186} C_VEL
LIN {X 0,Y 138.413,Z 564.424,A -85,B 0,C 180,E1 -28056.961,E2 -28056.961} C_VEL
LIN {X 0,Y 144.554,Z 552.038,A -85,B 0,C 180,E1 -28058.397,E2 -28058.397} C_VEL
LIN {X 0,Y 149.964,Z 538.206,A -85,B 0,C 180,E1 -28059.591,E2 -28059.591} C_VEL
LIN {X 0,Y 154.128,Z 524.147,A -85,B 0,C 180,E1 -28060.409,E2 -28060.409} C_VEL
LIN {X 0,Y 156.964,Z 510.289,A -85,B 0,C 180,E1 -28060.938,E2 -28060.938} C_VEL
LIN {X 0,Y 159.635,Z 487.099,A -85,B 0,C 180,E1 -28061.559,E2 -28061.559} C_VEL
LIN {X 0,Y 157.315,Z 481.21,A -85,B 0,C 180,E1 -28065.288,E2 -28065.288} C_VEL
LIN {X 0,Y 155.353,Z 476.695,A -85,B 0,C 180,E1 -28069.41,E2 -28069.41} C_VEL
LIN {X 0,Y 154.217,Z 473.826,A -85,B 0,C 180,E1 -28072.965,E2 -28072.965} C_VEL
LIN {X 0,Y 153.436,Z 470.668,A -85,B 0,C 180,E1 -28080,E2 -28080} C_VEL
LIN {X 0,Y 154.483,Z 474.465,A -85,B 0,C 180,E1 -28088.05,E2 -28088.05} C_VEL
LIN {X 0,Y 155.894,Z 477.978,A -85,B 0,C 180,E1 -28091.931,E2 -28091.931} C_VEL
LIN {X 0,Y 157.742,Z 482.215,A -85,B 0,C 180,E1 -28095.505,E2 -28095.505} C_VEL
LIN {X 0,Y 159.642,Z 487.127,A -85,B 0,C 180,E1 -28098.497,E2 -28098.497} C_VEL
LIN {X 0,Y 156.766,Z 511.434,A -85,B 0,C 180,E1 -28099.145,E2 -28099.145} C_VEL
LIN {X 0,Y 153.636,Z 526.181,A -85,B 0,C 180,E1 -28099.772,E2 -28099.772} C_VEL
LIN {X 0,Y 149.242,Z 540.359,A -85,B 0,C 180,E1 -28100.63,E2 -28100.63} C_VEL
LIN {X 0,Y 143.802,Z 553.72,A -85,B 0,C 180,E1 -28101.796,E2 -28101.796} C_VEL
LIN {X 0,Y 137.688,Z 565.771,A -85,B 0,C 180,E1 -28103.263,E2 -28103.263} C_VEL
LIN {X 0,Y 130.026,Z 578.148,A -85,B 0,C 180,E1 -28105.322,E2 -28105.322} C_VEL
LIN {X 0,Y 122.844,Z 588.071,A -85,B 0,C 180,E1 -28107.623,E2 -28107.623} C_VEL
LIN {X 0,Y 114.375,Z 597.983,A -85,B 0,C 180,E1 -28110.664,E2 -28110.664} C_VEL
LIN {X 0,Y 106.199,Z 606.282,A -85,B 0,C 180,E1 -28114.195,E2 -28114.195} C_VEL
LIN {X 0,Y 97.274,Z 614.215,A -85,B 0,C 180,E1 -28119.051,E2 -28119.051} C_VEL
LIN {X 0,Y 89.219,Z 620.596,A -85,B 0,C 180,E1 -28124.859,E2 -28124.859} C_VEL
LIN {X 0,Y 83.231,Z 625.013,A -85,B 0,C 180,E1 -28130.715,E2 -28130.715} C_VEL
LIN {X 0,Y 78.095,Z 628.492,A -85,B 0,C 180,E1 -28137.327,E2 -28137.327} C_VEL
LIN {X 0,Y 72.952,Z 631.867,A -85,B 0,C 180,E1 -28147.342,E2 -28147.342} C_VEL
LIN {X 0,Y 70.194,Z 633.853,A -85,B 0,C 180,E1 -28158.456,E2 -28158.456} C_VEL
LIN {X 0,Y 69.648,Z 634.342,A -85,B 0,C 180,E1 -28164.216,E2 -28164.216} C_VEL
LIN {X 0,Y 69.581,Z 634.5,A -85,B 0,C 180,E1 -28170.007,E2 -28170.007} C_VEL
LIN {X 0,Y 70.295,Z 633.819,A -85,B 0,C 180,E1 -28181.542,E2 -28181.542} C_VEL
LIN {X 0,Y 73.454,Z 631.8,A -85,B 0,C 180,E1 -28192.509,E2 -28192.509} C_VEL
LIN {X 0,Y 79.038,Z 628.397,A -85,B 0,C 180,E1 -28202.251,E2 -28202.251} C_VEL
LIN {X 0,Y 84.725,Z 624.907,A -85,B 0,C 180,E1 -28208.479,E2 -28208.479} C_VEL
LIN {X 0,Y 93.738,Z 619.038,A -85,B 0,C 180,E1 -28215.012,E2 -28215.012} C_VEL
LIN {X 0,Y 95.192,Z 618.025,A -85,B 0,C 180,E1 -28215.815,E2 -28215.815} C_VEL
LIN {X 0,Y 93.85,Z 617.458,A -85,B 0,C 180,E1 -28217.626,E2 -28217.626} C_VEL
LIN {X 0,Y 88.691,Z 616.974,A -85,B 0,C 180,E1 -28222.42,E2 -28222.42} C_VEL
LIN {X 0,Y 84.13,Z 615.616,A -85,B 0,C 180,E1 -28229.919,E2 -28229.919} C_VEL
LIN {X 0,Y 81.813,Z 614.994,A -85,B 0,C 180,E1 -28234.564,E2 -28234.564} C_VEL
LIN {X 0,Y 80.76,Z 614.23,A -85,B 0,C 180,E1 -28238.638,E2 -28238.638} C_VEL
LIN {X 0,Y 79.579,Z 613.776,A -85,B 0,C 180,E1 -28242.755,E2 -28242.755} C_VEL
LIN {X 0,Y 77.014,Z 613.899,A -85,B 0,C 180,E1 -28249.749,E2 -28249.749} C_VEL
LIN {X 0,Y 75.4,Z 614.128,A -85,B 0,C 180,E1 -28258.646,E2 -28258.646} C_VEL
LIN {X 0,Y 75.784,Z 613.913,A -85,B 0,C 180,E1 -28261.632,E2 -28261.632} C_VEL
LIN {X 0,Y 81.457,Z 612.165,A -85,B 0,C 180,E1 -28275.001,E2 -28275.001} C_VEL
LIN {X 0,Y 92.975,Z 609.504,A -85,B 0,C 180,E1 -28286.972,E2 -28286.972} C_VEL
LIN {X 0,Y 97.826,Z 608.349,A -85,B 0,C 180,E1 -28290.192,E2 -28290.192} C_VEL
LIN {X 0,Y 99.645,Z 608.496,A -85,B 0,C 180,E1 -28292.173,E2 -28292.173} C_VEL
LIN {X 0,Y 91.706,Z 615.02,A -85,B 0,C 180,E1 -28296.412,E2 -28296.412} C_VEL
LIN {X 0,Y 84.346,Z 620.436,A -85,B 0,C 180,E1 -28301.409,E2 -28301.409} C_VEL
LIN {X 0,Y 77.834,Z 624.889,A -85,B 0,C 180,E1 -28307.366,E2 -28307.366} C_VEL
LIN {X 0,Y 72.215,Z 628.383,A -85,B 0,C 180,E1 -28314.265,E2 -28314.265} C_VEL
LIN {X 0,Y 66.443,Z 631.79,A -85,B 0,C 180,E1 -28324.961,E2 -28324.961} C_VEL
LIN {X 0,Y 63.239,Z 633.813,A -85,B 0,C 180,E1 -28337.15,E2 -28337.15} C_VEL
LIN {X 0,Y 62.5,Z 634.499,A -85,B 0,C 180,E1 -28349.992,E2 -28349.992} C_VEL
LIN {X 0,Y 62.577,Z 634.344,A -85,B 0,C 180,E1 -28356.44,E2 -28356.44} C_VEL
LIN {X 0,Y 64.479,Z 633.037,A -85,B 0,C 180,E1 -28369.078,E2 -28369.078} C_VEL
LIN {X 0,Y 68.967,Z 630.371,A -85,B 0,C 180,E1 -28380.623,E2 -28380.623} C_VEL
LIN {X 0,Y 75.805,Z 626.272,A -85,B 0,C 180,E1 -28390.455,E2 -28390.455} C_VEL
LIN {X 0,Y 84.331,Z 620.618,A -85,B 0,C 180,E1 -28398.585,E2 -28398.585} C_VEL
LIN {X 0,Y 92.928,Z 614.241,A -85,B 0,C 180,E1 -28404.381,E2 -28404.381} C_VEL
LIN {X 0,Y 102.31,Z 606.313,A -85,B 0,C 180,E1 -28409.157,E2 -28409.157} C_VEL
LIN {X 0,Y 110.868,Z 598.02,A -85,B 0,C 180,E1 -28412.546,E2 -28412.546} C_VEL
LIN {X 0,Y 119.917,Z 587.784,A -85,B 0,C 180,E1 -28415.555,E2 -28415.555} C_VEL
LIN {X 0,Y 128.021,Z 576.905,A -85,B 0,C 180,E1 -28417.867,E2 -28417.867} C_VEL
LIN {X 0,Y 135.787,Z 564.419,A -85,B 0,C 180,E1 -28419.723,E2 -28419.723} C_VEL
LIN {X 0,Y 142.086,Z 552.033,A -85,B 0,C 180,E1 -28421.069,E2 -28421.069} C_VEL
LIN {X 0,Y 147.636,Z 538.198,A -85,B 0,C 180,E1 -28422.176,E2 -28422.176} C_VEL
LIN {X 0,Y 151.894,Z 524.137,A -85,B 0,C 180,E1 -28422.934,E2 -28422.934} C_VEL
LIN {X 0,Y 154.896,Z 509.742,A -85,B 0,C 180,E1 -28423.425,E2 -28423.425} C_VEL
LIN {X 0,Y 157.08,Z 491.11,A -85,B 0,C 180,E1 -28423.932,E2 -28423.932} C_VEL
LIN {X 0,Y 155.4,Z 486.54,A -85,B 0,C 180,E1 -28427.138,E2 -28427.138} C_VEL
LIN {X 0,Y 154.023,Z 483.101,A -85,B 0,C 180,E1 -28430.52,E2 -28430.52} C_VEL
LIN {X 0,Y 153.237,Z 480.787,A -85,B 0,C 180,E1 -28433.333,E2 -28433.333} C_VEL
LIN {X 0,Y 152.561,Z 477.79,A -85,B 0,C 180,E1 -28440,E2 -28440} C_VEL
LIN {X 0,Y 153.407,Z 481.255,A -85,B 0,C 180,E1 -28447.403,E2 -28447.403} C_VEL
LIN {X 0,Y 154.728,Z 484.907,A -85,B 0,C 180,E1 -28451.4,E2 -28451.4} C_VEL
LIN {X 0,Y 156.229,Z 488.68,A -85,B 0,C 180,E1 -28454.564,E2 -28454.564} C_VEL
LIN {X 0,Y 157.102,Z 491.148,A -85,B 0,C 180,E1 -28456.147,E2 -28456.147} C_VEL
LIN {X 0,Y 154.504,Z 511.921,A -85,B 0,C 180,E1 -28456.677,E2 -28456.677} C_VEL
LIN {X 0,Y 151.317,Z 526.44,A -85,B 0,C 180,E1 -28457.256,E2 -28457.256} C_VEL
LIN {X 0,Y 146.891,Z 540.366,A -85,B 0,C 180,E1 -28458.039,E2 -28458.039} C_VEL
LIN {X 0,Y 141.324,Z 553.725,A -85,B 0,C 180,E1 -28459.128,E2 -28459.128} C_VEL
LIN {X 0,Y 135.042,Z 565.775,A -85,B 0,C 180,E1 -28460.495,E2 -28460.495} C_VEL
LIN {X 0,Y 127.144,Z 578.152,A -85,B 0,C 180,E1 -28462.421,E2 -28462.421} C_VEL
LIN {X 0,Y 119.412,Z 588.429,A -85,B 0,C 180,E1 -28464.694,E2 -28464.694} C_VEL
LIN {X 0,Y 110.916,Z 597.986,A -85,B 0,C 180,E1 -28467.501,E2 -28467.501} C_VEL
LIN {X 0,Y 102.362,Z 606.284,A -85,B 0,C 180,E1 -28470.893,E2 -28470.893} C_VEL
LIN {X 0,Y 92.954,Z 614.217,A -85,B 0,C 180,E1 -28475.642,E2 -28475.642} C_VEL
LIN {X 0,Y 84.339,Z 620.598,A -85,B 0,C 180,E1 -28481.422,E2 -28481.422} C_VEL
LIN {X 0,Y 75.834,Z 626.256,A -85,B 0,C 180,E1 -28489.563,E2 -28489.563} C_VEL
LIN {X 0,Y 68.974,Z 630.359,A -85,B 0,C 180,E1 -28499.381,E2 -28499.381} C_VEL
LIN {X 0,Y 64.506,Z 633.03,A -85,B 0,C 180,E1 -28510.931,E2 -28510.931} C_VEL
LIN {X 0,Y 62.579,Z 634.342,A -85,B 0,C 180,E1 -28523.56,E2 -28523.56} C_VEL
LIN {X 0,Y 62.499,Z 634.5,A -85,B 0,C 180,E1 -28530.008,E2 -28530.008} C_VEL
LIN {X 0,Y 63.347,Z 633.818,A -85,B 0,C 180,E1 -28542.828,E2 -28542.828} C_VEL
LIN {X 0,Y 66.934,Z 631.8,A -85,B 0,C 180,E1 -28554.842,E2 -28554.842} C_VEL
LIN {X 0,Y 73.125,Z 628.397,A -85,B 0,C 180,E1 -28565.224,E2 -28565.224} C_VEL
LIN {X 0,Y 79.291,Z 624.906,A -85,B 0,C 180,E1 -28571.672,E2 -28571.672} C_VEL
LIN {X 0,Y 86.587,Z 620.457,A -85,B 0,C 180,E1 -28576.937,E2 -28576.937} C_VEL
LIN {X 0,Y 81.348,Z 619.755,A -85,B 0,C 180,E1 -28582.789,E2 -28582.789} C_VEL
LIN {X 0,Y 74.495,Z 617.523,A -85,B 0,C 180,E1 -28598.289,E2 -28598.289} C_VEL
LIN {X 0,Y 75.429,Z 614.099,A -85,B 0,C 180,E1 -28620,E2 -28620} C_VEL
LIN {X 0,Y 75.784,Z 613.913,A -85,B 0,C 180,E1 -28621.632,E2 -28621.632} C_VEL
LIN {X 0,Y 76.495,Z 613.73,A -85,B 0,C 180,E1 -28626.041,E2 -28626.041} C_VEL
LIN {X 0,Y 78.691,Z 614.708,A -85,B 0,C 180,E1 -28639.105,E2 -28639.105} C_VEL
LIN {X 0,Y 80.969,Z 614.604,A -85,B 0,C 180,E1 -28642.994,E2 -28642.994} C_VEL
LIN {X 0,Y 82.018,Z 614.43,A -85,B 0,C 180,E1 -28644.151,E2 -28644.151} C_VEL
LIN {X 0,Y 89.459,Z 613.006,A -85,B 0,C 180,E1 -28650.201,E2 -28650.201} C_VEL
LIN {X 0,Y 90.403,Z 613.005,A -85,B 0,C 180,E1 -28651.214,E2 -28651.214} C_VEL
LIN {X 0,Y 82.35,Z 618.762,A -85,B 0,C 180,E1 -28655.82,E2 -28655.82} C_VEL
LIN {X 0,Y 74.969,Z 623.489,A -85,B 0,C 180,E1 -28661.404,E2 -28661.404} C_VEL
LIN {X 0,Y 66.561,Z 628.383,A -85,B 0,C 180,E1 -28670.68,E2 -28670.68} C_VEL
LIN {X 0,Y 60.044,Z 631.79,A -85,B 0,C 180,E1 -28682.074,E2 -28682.074} C_VEL
LIN {X 0,Y 56.321,Z 633.813,A -85,B 0,C 180,E1 -28695.539,E2 -28695.539} C_VEL
LIN {X 0,Y 55.54,Z 634.322,A -85,B 0,C 180,E1 -28702.721,E2 -28702.721} C_VEL
LIN {X 0,Y 55.402,Z 634.499,A -85,B 0,C 180,E1 -28709.991,E2 -28709.991} C_VEL
LIN {X 0,Y 55.53,Z 634.344,A -85,B 0,C 180,E1 -28717.262,E2 -28717.262} C_VEL
LIN {X 0,Y 57.806,Z 633.037,A -85,B 0,C 180,E1 -28731.382,E2 -28731.382} C_VEL
LIN {X 0,Y 62.936,Z 630.37,A -85,B 0,C 180,E1 -28743.931,E2 -28743.931} C_VEL
LIN {X 0,Y 70.526,Z 626.271,A -85,B 0,C 180,E1 -28754.221,E2 -28754.221} C_VEL
LIN {X 0,Y 79.783,Z 620.616,A -85,B 0,C 180,E1 -28762.437,E2 -28762.437} C_VEL
LIN {X 0,Y 88.964,Z 614.239,A -85,B 0,C 180,E1 -28768.116,E2 -28768.116} C_VEL
LIN {X 0,Y 98.836,Z 606.311,A -85,B 0,C 180,E1 -28772.716,E2 -28772.716} C_VEL
LIN {X 0,Y 107.774,Z 598.017,A -85,B 0,C 180,E1 -28775.903,E2 -28775.903} C_VEL
LIN {X 0,Y 117.51,Z 587.366,A -85,B 0,C 180,E1 -28778.821,E2 -28778.821} C_VEL
LIN {X 0,Y 125.522,Z 576.901,A -85,B 0,C 180,E1 -28780.866,E2 -28780.866} C_VEL
LIN {X 0,Y 133.49,Z 564.415,A -85,B 0,C 180,E1 -28782.587,E2 -28782.587} C_VEL
LIN {X 0,Y 139.939,Z 552.027,A -85,B 0,C 180,E1 -28783.826,E2 -28783.826} C_VEL
LIN {X 0,Y 145.619,Z 538.191,A -85,B 0,C 180,E1 -28784.837,E2 -28784.837} C_VEL
LIN {X 0,Y 149.841,Z 524.596,A -85,B 0,C 180,E1 -28785.503,E2 -28785.503} C_VEL
LIN {X 0,Y 152.934,Z 510.207,A -85,B 0,C 180,E1 -28785.963,E2 -28785.963} C_VEL
LIN {X 0,Y 154.787,Z 495.268,A -85,B 0,C 180,E1 -28786.372,E2 -28786.372} C_VEL
LIN {X 0,Y 153.481,Z 491.539,A -85,B 0,C 180,E1 -28789.446,E2 -28789.446} C_VEL
LIN {X 0,Y 152.263,Z 487.749,A -85,B 0,C 180,E1 -28793.706,E2 -28793.706} C_VEL
LIN {X 0,Y 151.687,Z 484.913,A -85,B 0,C 180,E1 -28800,E2 -28800} C_VEL
LIN {X 0,Y 152.391,Z 488.251,A -85,B 0,C 180,E1 -28806.953,E2 -28806.953} C_VEL
LIN {X 0,Y 153.499,Z 491.627,A -85,B 0,C 180,E1 -28810.657,E2 -28810.657} C_VEL
LIN {X 0,Y 154.739,Z 495.113,A -85,B 0,C 180,E1 -28813.569,E2 -28813.569} C_VEL
LIN {X 0,Y 154.807,Z 495.345,A -85,B 0,C 180,E1 -28813.717,E2 -28813.717} C_VEL
LIN {X 0,Y 152.366,Z 513.32,A -85,B 0,C 180,E1 -28814.159,E2 -28814.159} C_VEL
LIN {X 0,Y 149.012,Z 527.791,A -85,B 0,C 180,E1 -28814.724,E2 -28814.724} C_VEL
LIN {X 0,Y 144.451,Z 541.498,A -85,B 0,C 180,E1 -28815.449,E2 -28815.449} C_VEL
LIN {X 0,Y 139.16,Z 553.731,A -85,B 0,C 180,E1 -28816.366,E2 -28816.366} C_VEL
LIN {X 0,Y 132.722,Z 565.779,A -85,B 0,C 180,E1 -28817.622,E2 -28817.622} C_VEL
LIN {X 0,Y 124.761,Z 577.941,A -85,B 0,C 180,E1 -28819.356,E2 -28819.356} C_VEL
LIN {X 0,Y 116.303,Z 588.791,A -85,B 0,C 180,E1 -28821.598,E2 -28821.598} C_VEL
LIN {X 0,Y 107.814,Z 597.988,A -85,B 0,C 180,E1 -28824.144,E2 -28824.144} C_VEL
LIN {X 0,Y 98.891,Z 606.286,A -85,B 0,C 180,E1 -28827.345,E2 -28827.345} C_VEL
LIN {X 0,Y 88.994,Z 614.218,A -85,B 0,C 180,E1 -28831.915,E2 -28831.915} C_VEL
LIN {X 0,Y 79.788,Z 620.599,A -85,B 0,C 180,E1 -28837.568,E2 -28837.568} C_VEL
LIN {X 0,Y 70.552,Z 626.257,A -85,B 0,C 180,E1 -28845.8,E2 -28845.8} C_VEL
LIN {X 0,Y 62.944,Z 630.36,A -85,B 0,C 180,E1 -28856.074,E2 -28856.074} C_VEL
LIN {X 0,Y 57.827,Z 633.03,A -85,B 0,C 180,E1 -28868.627,E2 -28868.627} C_VEL
LIN {X 0,Y 55.534,Z 634.342,A -85,B 0,C 180,E1 -28882.739,E2 -28882.739} C_VEL
LIN {X 0,Y 55.401,Z 634.5,A -85,B 0,C 180,E1 -28890.009,E2 -28890.009} C_VEL
LIN {X 0,Y 56.449,Z 633.818,A -85,B 0,C 180,E1 -28904.428,E2 -28904.428} C_VEL
LIN {X 0,Y 60.552,Z 631.799,A -85,B 0,C 180,E1 -28917.672,E2 -28917.672} C_VEL
LIN {X 0,Y 67.443,Z 628.396,A -85,B 0,C 180,E1 -28928.709,E2 -28928.709} C_VEL
LIN {X 0,Y 74.144,Z 624.905,A -85,B 0,C 180,E1 -28935.319,E2 -28935.319} C_VEL
LIN {X 0,Y 76.619,Z 623.505,A -85,B 0,C 180,E1 -28937.216,E2 -28937.216} C_VEL
LIN {X 0,Y 76.223,Z 622.699,A -85,B 0,C 180,E1 -28939.803,E2 -28939.803} C_VEL
LIN {X 0,Y 67.98,Z 620.451,A -85,B 0,C 180,E1 -28958.525,E2 -28958.525} C_VEL
LIN {X 0,Y 69.048,Z 617.601,A -85,B 0,C 180,E1 -28980,E2 -28980} C_VEL
LIN {X 0,Y 79.119,Z 615.01,A -85,B 0,C 180,E1 -29001.07,E2 -29001.07} C_VEL
LIN {X 0,Y 82.018,Z 614.43,A -85,B 0,C 180,E1 -29004.151,E2 -29004.151} C_VEL
LIN {X 0,Y 82.746,Z 614.615,A -85,B 0,C 180,E1 -29005.747,E2 -29005.747} C_VEL
LIN {X 0,Y 82.276,Z 615.686,A -85,B 0,C 180,E1 -29007.973,E2 -29007.973} C_VEL
LIN {X 0,Y 80.221,Z 617.658,A -85,B 0,C 180,E1 -29010.661,E2 -29010.661} C_VEL
LIN {X 0,Y 77.9,Z 619.338,A -85,B 0,C 180,E1 -29012.577,E2 -29012.577} C_VEL
LIN {X 0,Y 71.084,Z 623.303,A -85,B 0,C 180,E1 -29017.102,E2 -29017.102} C_VEL
LIN {X 0,Y 64.525,Z 626.707,A -85,B 0,C 180,E1 -29022.59,E2 -29022.59} C_VEL
LIN {X 0,Y 57.189,Z 630.266,A -85,B 0,C 180,E1 -29032.077,E2 -29032.077} C_VEL
LIN {X 0,Y 51.268,Z 632.971,A -85,B 0,C 180,E1 -29045.706,E2 -29045.706} C_VEL
LIN {X 0,Y 48.498,Z 634.323,A -85,B 0,C 180,E1 -29061.657,E2 -29061.657} C_VEL
LIN {X 0,Y 48.319,Z 634.499,A -85,B 0,C 180,E1 -29069.989,E2 -29069.989} C_VEL
LIN {X 0,Y 48.488,Z 634.344,A -85,B 0,C 180,E1 -29078.323,E2 -29078.323} C_VEL
LIN {X 0,Y 51.222,Z 633.036,A -85,B 0,C 180,E1 -29094.296,E2 -29094.296} C_VEL
LIN {X 0,Y 57.164,Z 630.369,A -85,B 0,C 180,E1 -29107.92,E2 -29107.92} C_VEL
LIN {X 0,Y 65.604,Z 626.27,A -85,B 0,C 180,E1 -29118.569,E2 -29118.569} C_VEL
LIN {X 0,Y 75.643,Z 620.615,A -85,B 0,C 180,E1 -29126.727,E2 -29126.727} C_VEL
LIN {X 0,Y 85.402,Z 614.238,A -85,B 0,C 180,E1 -29132.195,E2 -29132.195} C_VEL
LIN {X 0,Y 95.78,Z 606.309,A -85,B 0,C 180,E1 -29136.506,E2 -29136.506} C_VEL
LIN {X 0,Y 105.073,Z 598.015,A -85,B 0,C 180,E1 -29139.443,E2 -29139.443} C_VEL
LIN {X 0,Y 115.13,Z 587.363,A -85,B 0,C 180,E1 -29142.125,E2 -29142.125} C_VEL
LIN {X 0,Y 123.376,Z 576.897,A -85,B 0,C 180,E1 -29143.984,E2 -29143.984} C_VEL
LIN {X 0,Y 131.541,Z 564.41,A -85,B 0,C 180,E1 -29145.537,E2 -29145.537} C_VEL
LIN {X 0,Y 138.132,Z 552.021,A -85,B 0,C 180,E1 -29146.652,E2 -29146.652} C_VEL
LIN {X 0,Y 143.928,Z 538.184,A -85,B 0,C 180,E1 -29147.561,E2 -29147.561} C_VEL
LIN {X 0,Y 148.41,Z 523.912,A -85,B 0,C 180,E1 -29148.183,E2 -29148.183} C_VEL
LIN {X 0,Y 151.496,Z 509.521,A -85,B 0,C 180,E1 -29148.58,E2 -29148.58} C_VEL
LIN {X 0,Y 152.78,Z 499.749,A -85,B 0,C 180,E1 -29148.813,E2 -29148.813} C_VEL
LIN {X 0,Y 151.684,Z 496.372,A -85,B 0,C 180,E1 -29152.219,E2 -29152.219} C_VEL
LIN {X 0,Y 151.175,Z 494.461,A -85,B 0,C 180,E1 -29154.665,E2 -29154.665} C_VEL
LIN {X 0,Y 150.81,Z 492.057,A -85,B 0,C 180,E1 -29160,E2 -29160} C_VEL
LIN {X 0,Y 151.363,Z 495.114,A -85,B 0,C 180,E1 -29166.373,E2 -29166.373} C_VEL
LIN {X 0,Y 152.304,Z 498.393,A -85,B 0,C 180,E1 -29169.932,E2 -29169.932} C_VEL
LIN {X 0,Y 152.768,Z 499.724,A -85,B 0,C 180,E1 -29171.204,E2 -29171.204} C_VEL
LIN {X 0,Y 150.458,Z 515.174,A -85,B 0,C 180,E1 -29171.603,E2 -29171.603} C_VEL
LIN {X 0,Y 146.807,Z 529.712,A -85,B 0,C 180,E1 -29172.128,E2 -29172.128} C_VEL
LIN {X 0,Y 142.312,Z 542.531,A -85,B 0,C 180,E1 -29172.768,E2 -29172.768} C_VEL
LIN {X 0,Y 136.501,Z 555.355,A -85,B 0,C 180,E1 -29173.654,E2 -29173.654} C_VEL
LIN {X 0,Y 129.925,Z 567.088,A -85,B 0,C 180,E1 -29174.798,E2 -29174.798} C_VEL
LIN {X 0,Y 121.774,Z 579.013,A -85,B 0,C 180,E1 -29176.381,E2 -29176.381} C_VEL
LIN {X 0,Y 112.49,Z 590.34,A -85,B 0,C 180,E1 -29178.603,E2 -29178.603} C_VEL
LIN {X 0,Y 103.535,Z 599.475,A -85,B 0,C 180,E1 -29181.051,E2 -29181.051} C_VEL
LIN {X 0,Y 94.318,Z 607.519,A -85,B 0,C 180,E1 -29184.12,E2 -29184.12} C_VEL
LIN {X 0,Y 83.99,Z 615.227,A -85,B 0,C 180,E1 -29188.54,E2 -29188.54} C_VEL
LIN {X 0,Y 75.649,Z 620.6,A -85,B 0,C 180,E1 -29193.28,E2 -29193.28} C_VEL
LIN {X 0,Y 65.627,Z 626.258,A -85,B 0,C 180,E1 -29201.453,E2 -29201.453} C_VEL
LIN {X 0,Y 57.172,Z 630.36,A -85,B 0,C 180,E1 -29212.086,E2 -29212.086} C_VEL
LIN {X 0,Y 51.24,Z 633.031,A -85,B 0,C 180,E1 -29225.714,E2 -29225.714} C_VEL
LIN {X 0,Y 48.491,Z 634.342,A -85,B 0,C 180,E1 -29241.677,E2 -29241.677} C_VEL
LIN {X 0,Y 48.318,Z 634.5,A -85,B 0,C 180,E1 -29250.011,E2 -29250.011} C_VEL
LIN {X 0,Y 49.594,Z 633.818,A -85,B 0,C 180,E1 -29266.475,E2 -29266.475} C_VEL
LIN {X 0,Y 54.358,Z 631.798,A -85,B 0,C 180,E1 -29281.153,E2 -29281.153} C_VEL
LIN {X 0,Y 62.057,Z 628.395,A -85,B 0,C 180,E1 -29292.815,E2 -29292.815} C_VEL
LIN {X 0,Y 68.136,Z 625.481,A -85,B 0,C 180,E1 -29298.567,E2 -29298.567} C_VEL
LIN {X 0,Y 67.699,Z 624.815,A -85,B 0,C 180,E1 -29301.474,E2 -29301.474} C_VEL
LIN {X 0,Y 61.223,Z 622.996,A -85,B 0,C 180,E1 -29319.857,E2 -29319.857} C_VEL
LIN {X 0,Y 63.395,Z 620.446,A -85,B 0,C 180,E1 -29343.735,E2 -29343.735} C_VEL
LIN {X 0,Y 73.893,Z 618.304,A -85,B 0,C 180,E1 -29363.682,E2 -29363.682} C_VEL
LIN {X 0,Y 80.171,Z 617.25,A -85,B 0,C 180,E1 -29369.591,E2 -29369.591} C_VEL
LIN {X 0,Y 79.624,Z 617.955,A -85,B 0,C 180,E1 -29370.868,E2 -29370.868} C_VEL
LIN {X 0,Y 70.441,Z 623.49,A -85,B 0,C 180,E1 -29377.033,E2 -29377.033} C_VEL
LIN {X 0,Y 64.525,Z 626.707,A -85,B 0,C 180,E1 -29382.59,E2 -29382.59} C_VEL
LIN {X 0,Y 60.558,Z 628.493,A -85,B 0,C 180,E1 -29386.251,E2 -29386.251} C_VEL
LIN {X 0,Y 53.029,Z 630.902,A -85,B 0,C 180,E1 -29392.304,E2 -29392.304} C_VEL
LIN {X 0,Y 47.33,Z 632.384,A -85,B 0,C 180,E1 -29398.449,E2 -29398.449} C_VEL
LIN {X 0,Y 44.145,Z 633.26,A -85,B 0,C 180,E1 -29404.625,E2 -29404.625} C_VEL
LIN {X 0,Y 43.45,Z 633.466,A -85,B 0,C 180,E1 -29407.022,E2 -29407.022} C_VEL
LIN {X 0,Y 41.473,Z 634.323,A -85,B 0,C 180,E1 -29420.231,E2 -29420.231} C_VEL
LIN {X 0,Y 41.211,Z 634.499,A -85,B 0,C 180,E1 -29429.988,E2 -29429.988} C_VEL
LIN {X 0,Y 41.461,Z 634.344,A -85,B 0,C 180,E1 -29439.747,E2 -29439.747} C_VEL
LIN {X 0,Y 44.811,Z 633.036,A -85,B 0,C 180,E1 -29458.054,E2 -29458.054} C_VEL
LIN {X 0,Y 51.734,Z 630.369,A -85,B 0,C 180,E1 -29472.771,E2 -29472.771} C_VEL
LIN {X 0,Y 61.12,Z 626.269,A -85,B 0,C 180,E1 -29483.586,E2 -29483.586} C_VEL
LIN {X 0,Y 71.976,Z 620.614,A -85,B 0,C 180,E1 -29491.482,E2 -29491.482} C_VEL
LIN {X 0,Y 82.315,Z 614.236,A -85,B 0,C 180,E1 -29496.593,E2 -29496.593} C_VEL
LIN {X 0,Y 93.173,Z 606.307,A -85,B 0,C 180,E1 -29500.52,E2 -29500.52} C_VEL
LIN {X 0,Y 102.789,Z 598.012,A -85,B 0,C 180,E1 -29503.162,E2 -29503.162} C_VEL
LIN {X 0,Y 112.596,Z 587.967,A -85,B 0,C 180,E1 -29505.438,E2 -29505.438} C_VEL
LIN {X 0,Y 121.605,Z 576.894,A -85,B 0,C 180,E1 -29507.21,E2 -29507.21} C_VEL
LIN {X 0,Y 129.951,Z 564.405,A -85,B 0,C 180,E1 -29508.568,E2 -29508.568} C_VEL
LIN {X 0,Y 136.668,Z 552.016,A -85,B 0,C 180,E1 -29509.549,E2 -29509.549} C_VEL
LIN {X 0,Y 142.568,Z 538.177,A -85,B 0,C 180,E1 -29510.347,E2 -29510.347} C_VEL
LIN {X 0,Y 147.128,Z 523.886,A -85,B 0,C 180,E1 -29510.883,E2 -29510.883} C_VEL
LIN {X 0,Y 150.213,Z 509.722,A -85,B 0,C 180,E1 -29511.227,E2 -29511.227} C_VEL
LIN {X 0,Y 150.952,Z 504.537,A -85,B 0,C 180,E1 -29511.368,E2 -29511.368} C_VEL
LIN {X 0,Y 150.159,Z 501.216,A -85,B 0,C 180,E1 -29515.47,E2 -29515.47} C_VEL
LIN {X 0,Y 149.93,Z 499.218,A -85,B 0,C 180,E1 -29520,E2 -29520} C_VEL
LIN {X 0,Y 150.348,Z 502.006,A -85,B 0,C 180,E1 -29525.785,E2 -29525.785} C_VEL
LIN {X 0,Y 150.944,Z 504.56,A -85,B 0,C 180,E1 -29528.666,E2 -29528.666} C_VEL
LIN {X 0,Y 148.393,Z 518.78,A -85,B 0,C 180,E1 -29529.043,E2 -29529.043} C_VEL
LIN {X 0,Y 144.475,Z 532.816,A -85,B 0,C 180,E1 -29529.524,E2 -29529.524} C_VEL
LIN {X 0,Y 139.223,Z 546.514,A -85,B 0,C 180,E1 -29530.17,E2 -29530.17} C_VEL
LIN {X 0,Y 133.321,Z 558.523,A -85,B 0,C 180,E1 -29530.967,E2 -29530.967} C_VEL
LIN {X 0,Y 125.79,Z 570.964,A -85,B 0,C 180,E1 -29532.134,E2 -29532.134} C_VEL
LIN {X 0,Y 117.492,Z 582.212,A -85,B 0,C 180,E1 -29533.606,E2 -29533.606} C_VEL
LIN {X 0,Y 109.304,Z 591.562,A -85,B 0,C 180,E1 -29535.34,E2 -29535.34} C_VEL
LIN {X 0,Y 99.594,Z 600.96,A -85,B 0,C 180,E1 -29537.721,E2 -29537.721} C_VEL
LIN {X 0,Y 90.07,Z 608.752,A -85,B 0,C 180,E1 -29540.572,E2 -29540.572} C_VEL
LIN {X 0,Y 80.832,Z 615.228,A -85,B 0,C 180,E1 -29544.104,E2 -29544.104} C_VEL
LIN {X 0,Y 71.982,Z 620.601,A -85,B 0,C 180,E1 -29548.527,E2 -29548.527} C_VEL
LIN {X 0,Y 61.14,Z 626.259,A -85,B 0,C 180,E1 -29556.439,E2 -29556.439} C_VEL
LIN {X 0,Y 51.742,Z 630.361,A -85,B 0,C 180,E1 -29567.237,E2 -29567.237} C_VEL
LIN {X 0,Y 44.826,Z 633.031,A -85,B 0,C 180,E1 -29581.956,E2 -29581.956} C_VEL
LIN {X 0,Y 41.466,Z 634.343,A -85,B 0,C 180,E1 -29600.254,E2 -29600.254} C_VEL
LIN {X 0,Y 41.211,Z 634.499,A -85,B 0,C 180,E1 -29610.012,E2 -29610.012} C_VEL
LIN {X 0,Y 42.832,Z 633.817,A -85,B 0,C 180,E1 -29629.17,E2 -29629.17} C_VEL
LIN {X 0,Y 48.42,Z 631.798,A -85,B 0,C 180,E1 -29645.504,E2 -29645.504} C_VEL
LIN {X 0,Y 57.05,Z 628.394,A -85,B 0,C 180,E1 -29657.671,E2 -29657.671} C_VEL
LIN {X 0,Y 59.001,Z 627.585,A -85,B 0,C 180,E1 -29659.479,E2 -29659.479} C_VEL
LIN {X 0,Y 59.83,Z 626.842,A -85,B 0,C 180,E1 -29662.119,E2 -29662.119} C_VEL
LIN {X 0,Y 54.849,Z 625.636,A -85,B 0,C 180,E1 -29677.394,E2 -29677.394} C_VEL
LIN {X 0,Y 56.275,Z 623.497,A -85,B 0,C 180,E1 -29702.226,E2 -29702.226} C_VEL
LIN {X 0,Y 70.195,Z 621.093,A -85,B 0,C 180,E1 -29728.243,E2 -29728.243} C_VEL
LIN {X 0,Y 69.144,Z 622.053,A -85,B 0,C 180,E1 -29730.227,E2 -29730.227} C_VEL
LIN {X 0,Y 58.643,Z 627.322,A -85,B 0,C 180,E1 -29738.819,E2 -29738.819} C_VEL
LIN {X 0,Y 51.76,Z 630.266,A -85,B 0,C 180,E1 -29747.229,E2 -29747.229} C_VEL
LIN {X 0,Y 44.851,Z 632.971,A -85,B 0,C 180,E1 -29761.948,E2 -29761.948} C_VEL
LIN {X 0,Y 43.45,Z 633.466,A -85,B 0,C 180,E1 -29767.022,E2 -29767.022} C_VEL
LIN {X 0,Y 41.34,Z 634.064,A -85,B 0,C 180,E1 -29774.438,E2 -29774.438} C_VEL
LIN {X 0,Y 38.885,Z 634.385,A -85,B 0,C 180,E1 -29782.178,E2 -29782.178} C_VEL
LIN {X 0,Y 35.309,Z 634.37,A -85,B 0,C 180,E1 -29800.059,E2 -29800.059} C_VEL
LIN {X 0,Y 35.496,Z 634.008,A -85,B 0,C 180,E1 -29809.806,E2 -29809.806} C_VEL
LIN {X 0,Y 35.995,Z 633.859,A -85,B 0,C 180,E1 -29812.918,E2 -29812.918} C_VEL
LIN {X 0,Y 42.299,Z 631.875,A -85,B 0,C 180,E1 -29831.636,E2 -29831.636} C_VEL
LIN {X 0,Y 51.781,Z 628.504,A -85,B 0,C 180,E1 -29844.505,E2 -29844.505} C_VEL
LIN {X 0,Y 63.17,Z 623.5,A -85,B 0,C 180,E1 -29853.575,E2 -29853.575} C_VEL
LIN {X 0,Y 75.024,Z 617.15,A -85,B 0,C 180,E1 -29859.495,E2 -29859.495} C_VEL
LIN {X 0,Y 86.171,Z 609.922,A -85,B 0,C 180,E1 -29863.377,E2 -29863.377} C_VEL
LIN {X 0,Y 95.989,Z 602.346,A -85,B 0,C 180,E1 -29865.935,E2 -29865.935} C_VEL
LIN {X 0,Y 105.939,Z 593.253,A -85,B 0,C 180,E1 -29868.076,E2 -29868.076} C_VEL
LIN {X 0,Y 114.329,Z 584.192,A -85,B 0,C 180,E1 -29869.565,E2 -29869.565} C_VEL
LIN {X 0,Y 122.775,Z 573.38,A -85,B 0,C 180,E1 -29870.881,E2 -29870.881} C_VEL
LIN {X 0,Y 130.435,Z 561.55,A -85,B 0,C 180,E1 -29871.886,E2 -29871.886} C_VEL
LIN {X 0,Y 137.272,Z 548.477,A -85,B 0,C 180,E1 -29872.694,E2 -29872.694} C_VEL
LIN {X 0,Y 142.726,Z 535.051,A -85,B 0,C 180,E1 -29873.275,E2 -29873.275} C_VEL
LIN {X 0,Y 146.937,Z 520.938,A -85,B 0,C 180,E1 -29873.685,E2 -29873.685} C_VEL
LIN {X 0,Y 149.3,Z 509.582,A -85,B 0,C 180,E1 -29873.99,E2 -29873.99} C_VEL
LIN {X 0,Y 149.048,Z 507.98,A -85,B 0,C 180,E1 -29876.282,E2 -29876.282} C_VEL
LIN {X 0,Y 148.969,Z 506.345,A -85,B 0,C 180,E1 -29880,E2 -29880} C_VEL
LIN {X 0,Y 149.212,Z 508.885,A -85,B 0,C 180,E1 -29885.234,E2 -29885.234} C_VEL
LIN {X 0,Y 149.304,Z 509.566,A -85,B 0,C 180,E1 -29886.06,E2 -29886.06} C_VEL
LIN {X 0,Y 146.3,Z 523.452,A -85,B 0,C 180,E1 -29886.434,E2 -29886.434} C_VEL
LIN {X 0,Y 142.156,Z 536.606,A -85,B 0,C 180,E1 -29886.838,E2 -29886.838} C_VEL
LIN {X 0,Y 136.43,Z 550.216,A -85,B 0,C 180,E1 -29887.447,E2 -29887.447} C_VEL
LIN {X 0,Y 129.601,Z 562.952,A -85,B 0,C 180,E1 -29888.277,E2 -29888.277} C_VEL
LIN {X 0,Y 121.942,Z 574.533,A -85,B 0,C 180,E1 -29889.285,E2 -29889.285} C_VEL
LIN {X 0,Y 113.27,Z 585.414,A -85,B 0,C 180,E1 -29890.644,E2 -29890.644} C_VEL
LIN {X 0,Y 104.313,Z 594.863,A -85,B 0,C 180,E1 -29892.358,E2 -29892.358} C_VEL
LIN {X 0,Y 94.355,Z 603.686,A -85,B 0,C 180,E1 -29894.489,E2 -29894.489} C_VEL
LIN {X 0,Y 82.974,Z 612.141,A -85,B 0,C 180,E1 -29897.679,E2 -29897.679} C_VEL
LIN {X 0,Y 71.922,Z 618.948,A -85,B 0,C 180,E1 -29901.848,E2 -29901.848} C_VEL
LIN {X 0,Y 62.87,Z 623.635,A -85,B 0,C 180,E1 -29906.601,E2 -29906.601} C_VEL
LIN {X 0,Y 51.796,Z 628.497,A -85,B 0,C 180,E1 -29915.518,E2 -29915.518} C_VEL
LIN {X 0,Y 42.303,Z 631.87,A -85,B 0,C 180,E1 -29928.369,E2 -29928.369} C_VEL
LIN {X 0,Y 36.018,Z 633.854,A -85,B 0,C 180,E1 -29947.045,E2 -29947.045} C_VEL
LIN {X 0,Y 34.487,Z 634.343,A -85,B 0,C 180,E1 -29958.257,E2 -29958.257} C_VEL
LIN {X 0,Y 34.105,Z 634.499,A -85,B 0,C 180,E1 -29970.015,E2 -29970.015} C_VEL
LIN {X 0,Y 36.208,Z 633.817,A -85,B 0,C 180,E1 -29992.857,E2 -29992.857} C_VEL
LIN {X 0,Y 42.842,Z 631.797,A -85,B 0,C 180,E1 -30011.024,E2 -30011.024} C_VEL
LIN {X 0,Y 51.162,Z 628.94,A -85,B 0,C 180,E1 -30022.077,E2 -30022.077} C_VEL
LIN {X 0,Y 50.452,Z 628.393,A -85,B 0,C 180,E1 -30026.717,E2 -30026.717} C_VEL
LIN {X 0,Y 50.893,Z 625.713,A -85,B 0,C 180,E1 -30067.938,E2 -30067.938} C_VEL
LIN {X 0,Y 60.991,Z 624.346,A -85,B 0,C 180,E1 -30087.447,E2 -30087.447} C_VEL
LIN {X 0,Y 54.443,Z 627.323,A -85,B 0,C 180,E1 -30092.941,E2 -30092.941} C_VEL
LIN {X 0,Y 46.788,Z 630.267,A -85,B 0,C 180,E1 -30101.302,E2 -30101.302} C_VEL
LIN {X 0,Y 38.699,Z 632.972,A -85,B 0,C 180,E1 -30116.972,E2 -30116.972} C_VEL
LIN {X 0,Y 34.495,Z 634.323,A -85,B 0,C 180,E1 -30138.229,E2 -30138.229} C_VEL
LIN {X 0,Y 34.106,Z 634.499,A -85,B 0,C 180,E1 -30149.985,E2 -30149.985} C_VEL
LIN {X 0,Y 34.483,Z 634.344,A -85,B 0,C 180,E1 -30161.745,E2 -30161.745} C_VEL
LIN {X 0,Y 35.995,Z 633.859,A -85,B 0,C 180,E1 -30172.918,E2 -30172.918} C_VEL
LIN {X 0,Y 37.573,Z 633.319,A -85,B 0,C 180,E1 -30181.738,E2 -30181.738} C_VEL
LIN {X 0,Y 40.233,Z 631.886,A -85,B 0,C 180,E1 -30195.671,E2 -30195.671} C_VEL
LIN {X 0,Y 43.618,Z 630.256,A -85,B 0,C 180,E1 -30205.294,E2 -30205.294} C_VEL
LIN {X 0,Y 47.341,Z 628.756,A -85,B 0,C 180,E1 -30210.8,E2 -30210.8} C_VEL
LIN {X 0,Y 48.827,Z 628.189,A -85,B 0,C 180,E1 -30212.205,E2 -30212.205} C_VEL
LIN {X 0,Y 60.011,Z 623.643,A -85,B 0,C 180,E1 -30219.511,E2 -30219.511} C_VEL
LIN {X 0,Y 72.828,Z 617.149,A -85,B 0,C 180,E1 -30224.771,E2 -30224.771} C_VEL
LIN {X 0,Y 84.405,Z 609.92,A -85,B 0,C 180,E1 -30228.027,E2 -30228.027} C_VEL
LIN {X 0,Y 94.509,Z 602.344,A -85,B 0,C 180,E1 -30230.134,E2 -30230.134} C_VEL
LIN {X 0,Y 104.7,Z 593.25,A -85,B 0,C 180,E1 -30231.89,E2 -30231.89} C_VEL
LIN {X 0,Y 114.969,Z 582.23,A -85,B 0,C 180,E1 -30233.346,E2 -30233.346} C_VEL
LIN {X 0,Y 123.581,Z 570.986,A -85,B 0,C 180,E1 -30234.346,E2 -30234.346} C_VEL
LIN {X 0,Y 131.355,Z 558.548,A -85,B 0,C 180,E1 -30235.161,E2 -30235.161} C_VEL
LIN {X 0,Y 137.418,Z 546.545,A -85,B 0,C 180,E1 -30235.725,E2 -30235.725} C_VEL
LIN {X 0,Y 142.291,Z 534.383,A -85,B 0,C 180,E1 -30236.137,E2 -30236.137} C_VEL
LIN {X 0,Y 146.545,Z 520.015,A -85,B 0,C 180,E1 -30236.456,E2 -30236.456} C_VEL
LIN {X 0,Y 147.711,Z 514.875,A -85,B 0,C 180,E1 -30236.633,E2 -30236.633} C_VEL
LIN {X 0,Y 147.735,Z 513.41,A -85,B 0,C 180,E1 -30240,E2 -30240} C_VEL
LIN {X 0,Y 147.706,Z 514.929,A -85,B 0,C 180,E1 -30243.445,E2 -30243.445} C_VEL
LIN {X 0,Y 144.089,Z 529.003,A -85,B 0,C 180,E1 -30243.796,E2 -30243.796} C_VEL
LIN {X 0,Y 139.164,Z 542.55,A -85,B 0,C 180,E1 -30244.186,E2 -30244.186} C_VEL
LIN {X 0,Y 133.093,Z 555.37,A -85,B 0,C 180,E1 -30244.711,E2 -30244.711} C_VEL
LIN {X 0,Y 126.177,Z 567.1,A -85,B 0,C 180,E1 -30245.408,E2 -30245.408} C_VEL
LIN {X 0,Y 117.553,Z 579.024,A -85,B 0,C 180,E1 -30246.357,E2 -30246.357} C_VEL
LIN {X 0,Y 107.574,Z 590.369,A -85,B 0,C 180,E1 -30247.749,E2 -30247.749} C_VEL
LIN {X 0,Y 97.918,Z 599.482,A -85,B 0,C 180,E1 -30249.32,E2 -30249.32} C_VEL
LIN {X 0,Y 87.774,Z 607.525,A -85,B 0,C 180,E1 -30251.263,E2 -30251.263} C_VEL
LIN {X 0,Y 76.124,Z 615.231,A -85,B 0,C 180,E1 -30254.24,E2 -30254.24} C_VEL
LIN {X 0,Y 66.355,Z 620.604,A -85,B 0,C 180,E1 -30257.62,E2 -30257.62} C_VEL
LIN {X 0,Y 56.675,Z 625.125,A -85,B 0,C 180,E1 -30262.398,E2 -30262.398} C_VEL
LIN {X 0,Y 47.992,Z 628.498,A -85,B 0,C 180,E1 -30268.544,E2 -30268.544} C_VEL
LIN {X 0,Y 37.271,Z 631.87,A -85,B 0,C 180,E1 -30281.061,E2 -30281.061} C_VEL
LIN {X 0,Y 29.598,Z 633.855,A -85,B 0,C 180,E1 -30301.668,E2 -30301.668} C_VEL
LIN {X 0,Y 27.556,Z 634.343,A -85,B 0,C 180,E1 -30315.243,E2 -30315.243} C_VEL
LIN {X 0,Y 27.014,Z 634.499,A -85,B 0,C 180,E1 -30330.019,E2 -30330.019} C_VEL
LIN {X 0,Y 29.779,Z 633.817,A -85,B 0,C 180,E1 -30358.184,E2 -30358.184} C_VEL
LIN {X 0,Y 37.779,Z 631.797,A -85,B 0,C 180,E1 -30378.102,E2 -30378.102} C_VEL
LIN {X 0,Y 42.941,Z 630.273,A -85,B 0,C 180,E1 -30384.939,E2 -30384.939} C_VEL
LIN {X 0,Y 42.296,Z 629.887,A -85,B 0,C 180,E1 -30390.101,E2 -30390.101} C_VEL
LIN {X 0,Y 44.074,Z 627.985,A -85,B 0,C 180,E1 -30429.176,E2 -30429.176} C_VEL
LIN {X 0,Y 50.624,Z 627.223,A -85,B 0,C 180,E1 -30444.614,E2 -30444.614} C_VEL
LIN {X 0,Y 48.008,Z 628.387,A -85,B 0,C 180,E1 -30448.534,E2 -30448.534} C_VEL
LIN {X 0,Y 37.289,Z 631.793,A -85,B 0,C 180,E1 -30461.05,E2 -30461.05} C_VEL
LIN {X 0,Y 29.615,Z 633.814,A -85,B 0,C 180,E1 -30481.646,E2 -30481.646} C_VEL
LIN {X 0,Y 27.564,Z 634.323,A -85,B 0,C 180,E1 -30495.209,E2 -30495.209} C_VEL
LIN {X 0,Y 27.015,Z 634.499,A -85,B 0,C 180,E1 -30509.981,E2 -30509.981} C_VEL
LIN {X 0,Y 29.34,Z 633.901,A -85,B 0,C 180,E1 -30537.207,E2 -30537.207} C_VEL
LIN {X 0,Y 37.267,Z 631.874,A -85,B 0,C 180,E1 -30558.946,E2 -30558.946} C_VEL
LIN {X 0,Y 47.979,Z 628.503,A -85,B 0,C 180,E1 -30571.485,E2 -30571.485} C_VEL
LIN {X 0,Y 48.827,Z 628.189,A -85,B 0,C 180,E1 -30572.205,E2 -30572.205} C_VEL
LIN {X 0,Y 53.154,Z 626.464,A -85,B 0,C 180,E1 -30576.294,E2 -30576.294} C_VEL
LIN {X 0,Y 59.744,Z 623.324,A -85,B 0,C 180,E1 -30583.147,E2 -30583.147} C_VEL
LIN {X 0,Y 66.792,Z 619.627,A -85,B 0,C 180,E1 -30588.511,E2 -30588.511} C_VEL
LIN {X 0,Y 71.565,Z 616.99,A -85,B 0,C 180,E1 -30590.384,E2 -30590.384} C_VEL
LIN {X 0,Y 83.219,Z 609.919,A -85,B 0,C 180,E1 -30592.836,E2 -30592.836} C_VEL
LIN {X 0,Y 95.281,Z 600.972,A -85,B 0,C 180,E1 -30594.665,E2 -30594.665} C_VEL
LIN {X 0,Y 105.673,Z 591.576,A -85,B 0,C 180,E1 -30595.955,E2 -30595.955} C_VEL
LIN {X 0,Y 115.233,Z 581.171,A -85,B 0,C 180,E1 -30596.989,E2 -30596.989} C_VEL
LIN {X 0,Y 123.957,Z 569.691,A -85,B 0,C 180,E1 -30597.714,E2 -30597.714} C_VEL
LIN {X 0,Y 130.947,Z 558.543,A -85,B 0,C 180,E1 -30598.26,E2 -30598.26} C_VEL
LIN {X 0,Y 137.072,Z 546.539,A -85,B 0,C 180,E1 -30598.683,E2 -30598.683} C_VEL
LIN {X 0,Y 142.144,Z 533.916,A -85,B 0,C 180,E1 -30599,E2 -30599} C_VEL
LIN {X 0,Y 146.101,Z 520.735,A -85,B 0,C 180,E1 -30599.268,E2 -30599.268} C_VEL
LIN {X 0,Y 146.154,Z 520.46,A -85,B 0,C 180,E1 -30600,E2 -30600} C_VEL
LIN {X 0,Y 146.091,Z 520.779,A -85,B 0,C 180,E1 -30600.803,E2 -30600.803} C_VEL
LIN {X 0,Y 141.668,Z 535.319,A -85,B 0,C 180,E1 -30601.096,E2 -30601.096} C_VEL
LIN {X 0,Y 136.2,Z 548.46,A -85,B 0,C 180,E1 -30601.433,E2 -30601.433} C_VEL
LIN {X 0,Y 129.201,Z 561.536,A -85,B 0,C 180,E1 -30601.906,E2 -30601.906} C_VEL
LIN {X 0,Y 121.34,Z 573.367,A -85,B 0,C 180,E1 -30602.519,E2 -30602.519} C_VEL
LIN {X 0,Y 112.629,Z 584.18,A -85,B 0,C 180,E1 -30603.334,E2 -30603.334} C_VEL
LIN {X 0,Y 102.215,Z 594.868,A -85,B 0,C 180,E1 -30604.529,E2 -30604.529} C_VEL
LIN {X 0,Y 91.834,Z 603.69,A -85,B 0,C 180,E1 -30605.859,E2 -30605.859} C_VEL
LIN {X 0,Y 81.524,Z 611.029,A -85,B 0,C 180,E1 -30607.576,E2 -30607.576} C_VEL
LIN {X 0,Y 71.297,Z 617.143,A -85,B 0,C 180,E1 -30609.733,E2 -30609.733} C_VEL
LIN {X 0,Y 57.907,Z 623.637,A -85,B 0,C 180,E1 -30613.886,E2 -30613.886} C_VEL
LIN {X 0,Y 45.014,Z 628.498,A -85,B 0,C 180,E1 -30620.519,E2 -30620.519} C_VEL
LIN {X 0,Y 33.026,Z 631.871,A -85,B 0,C 180,E1 -30631.686,E2 -30631.686} C_VEL
LIN {X 0,Y 23.563,Z 633.855,A -85,B 0,C 180,E1 -30653.405,E2 -30653.405} C_VEL
LIN {X 0,Y 20.764,Z 634.343,A -85,B 0,C 180,E1 -30670.242,E2 -30670.242} C_VEL
LIN {X 0,Y 19.933,Z 634.499,A -85,B 0,C 180,E1 -30690.026,E2 -30690.026} C_VEL
LIN {X 0,Y 23.754,Z 633.816,A -85,B 0,C 180,E1 -30726.306,E2 -30726.306} C_VEL
LIN {X 0,Y 33.453,Z 631.796,A -85,B 0,C 180,E1 -30747.203,E2 -30747.203} C_VEL
LIN {X 0,Y 34.533,Z 631.521,A -85,B 0,C 180,E1 -30748.533,E2 -30748.533} C_VEL
LIN {X 0,Y 34.739,Z 631.245,A -85,B 0,C 180,E1 -30752.412,E2 -30752.412} C_VEL
LIN {X 0,Y 37.177,Z 629.925,A -85,B 0,C 180,E1 -30790.898,E2 -30790.898} C_VEL
LIN {X 0,Y 41.018,Z 629.526,A -85,B 0,C 180,E1 -30801.843,E2 -30801.843} C_VEL
LIN {X 0,Y 40.037,Z 629.927,A -85,B 0,C 180,E1 -30804.284,E2 -30804.284} C_VEL
LIN {X 0,Y 33.044,Z 631.793,A -85,B 0,C 180,E1 -30811.68,E2 -30811.68} C_VEL
LIN {X 0,Y 23.58,Z 633.815,A -85,B 0,C 180,E1 -30833.383,E2 -30833.383} C_VEL
LIN {X 0,Y 20.774,Z 634.323,A -85,B 0,C 180,E1 -30850.2,E2 -30850.2} C_VEL
LIN {X 0,Y 19.934,Z 634.499,A -85,B 0,C 180,E1 -30869.974,E2 -30869.974} C_VEL
LIN {X 0,Y 20.76,Z 634.344,A -85,B 0,C 180,E1 -30889.762,E2 -30889.762} C_VEL
LIN {X 0,Y 27.829,Z 633.035,A -85,B 0,C 180,E1 -30919.227,E2 -30919.227} C_VEL
LIN {X 0,Y 38.848,Z 630.366,A -85,B 0,C 180,E1 -30934.732,E2 -30934.732} C_VEL
LIN {X 0,Y 51.388,Z 626.266,A -85,B 0,C 180,E1 -30943.167,E2 -30943.167} C_VEL
LIN {X 0,Y 61.214,Z 622.213,A -85,B 0,C 180,E1 -30947.353,E2 -30947.353} C_VEL
LIN {X 0,Y 71.565,Z 616.99,A -85,B 0,C 180,E1 -30950.384,E2 -30950.384} C_VEL
LIN {X 0,Y 76.341,Z 614.211,A -85,B 0,C 180,E1 -30951.996,E2 -30951.996} C_VEL
LIN {X 0,Y 83.67,Z 609.434,A -85,B 0,C 180,E1 -30955.38,E2 -30955.38} C_VEL
LIN {X 0,Y 90.906,Z 604.168,A -85,B 0,C 180,E1 -30958.163,E2 -30958.163} C_VEL
LIN {X 0,Y 95.371,Z 600.558,A -85,B 0,C 180,E1 -30958.987,E2 -30958.987} C_VEL
LIN {X 0,Y 105.411,Z 591.573,A -85,B 0,C 180,E1 -30959.812,E2 -30959.812} C_VEL
LIN {X 0,Y 107.634,Z 589.319,A -85,B 0,C 180,E1 -30960,E2 -30960} C_VEL
LIN {X 0,Y 98.392,Z 598.002,A -85,B 0,C 180,E1 -30960.814,E2 -30960.814} C_VEL
LIN {X 0,Y 87.88,Z 606.298,A -85,B 0,C 180,E1 -30961.734,E2 -30961.734} C_VEL
LIN {X 0,Y 75.661,Z 614.228,A -85,B 0,C 180,E1 -30963.221,E2 -30963.221} C_VEL
LIN {X 0,Y 63.511,Z 620.607,A -85,B 0,C 180,E1 -30965.266,E2 -30965.266} C_VEL
LIN {X 0,Y 54.345,Z 624.58,A -85,B 0,C 180,E1 -30967.43,E2 -30967.43} C_VEL
LIN {X 0,Y 43.033,Z 628.499,A -85,B 0,C 180,E1 -30971.567,E2 -30971.567} C_VEL
LIN {X 0,Y 29.901,Z 631.871,A -85,B 0,C 180,E1 -30979.97,E2 -30979.97} C_VEL
LIN {X 0,Y 18.342,Z 633.855,A -85,B 0,C 180,E1 -31000.018,E2 -31000.018} C_VEL
LIN {X 0,Y 12.838,Z 634.499,A -85,B 0,C 180,E1 -31050.04,E2 -31050.04} C_VEL
LIN {X 0,Y 18.518,Z 633.816,A -85,B 0,C 180,E1 -31099.422,E2 -31099.422} C_VEL
LIN {X 0,Y 26.117,Z 632.587,A -85,B 0,C 180,E1 -31114.213,E2 -31114.213} C_VEL
LIN {X 0,Y 26.874,Z 632.199,A -85,B 0,C 180,E1 -31124.841,E2 -31124.841} C_VEL
LIN {X 0,Y 30.981,Z 631.456,A -85,B 0,C 180,E1 -31156.162,E2 -31156.162} C_VEL
LIN {X 0,Y 29.92,Z 631.794,A -85,B 0,C 180,E1 -31159.97,E2 -31159.97} C_VEL
